C05456=1021.407,257.153,370.993,169.626,49.435,159.469
C05457=1021.401,256.905,371.022,169.622,49.439,159.470
C05458=1021.394,256.657,371.050,169.618,49.443,159.470
C05459=1021.388,256.409,371.079,169.613,49.447,159.470
C05460=1021.381,256.160,371.108,169.610,49.452,159.470
C05461=1021.375,255.912,371.135,169.605,49.456,159.471
C05462=1021.369,255.664,371.165,169.601,49.460,159.471
C05463=1021.362,255.416,371.194,169.596,49.464,159.471
C05464=1021.356,255.167,371.221,169.592,49.469,159.471
C05465=1021.349,254.919,371.250,169.588,49.473,159.472
C05466=1021.343,254.670,371.279,169.583,49.477,159.472
C05467=1021.337,254.422,371.308,169.580,49.481,159.472
C05468=1021.330,254.174,371.335,169.575,49.486,159.473
C05469=1021.324,253.926,371.364,169.571,49.490,159.473
C05470=1021.318,253.677,371.393,169.567,49.494,159.473
C05471=1021.311,253.429,371.421,169.563,49.499,159.474
C05472=1021.305,253.180,371.450,169.559,49.503,159.474
C05473=1021.299,252.932,371.479,169.555,49.507,159.474
C05474=1021.292,252.684,371.506,169.550,49.511,159.474
C05475=1021.286,252.436,371.535,169.546,49.516,159.475
C05476=1021.280,252.187,371.564,169.542,49.520,159.475
C05477=1021.273,251.939,371.592,169.538,49.524,159.475
C05478=1021.267,251.690,371.620,169.534,49.529,159.476
C05479=1021.262,251.442,371.648,169.530,49.533,159.476
C05480=1021.255,251.195,371.677,169.525,49.538,159.476
C05481=1021.249,250.946,371.705,169.522,49.542,159.477
C05482=1021.243,250.698,371.734,169.517,49.547,159.477
C05483=1021.236,250.449,371.762,169.513,49.551,159.477
C05484=1021.230,250.200,371.790,169.509,49.555,159.477
C05485=1021.224,249.952,371.819,169.504,49.560,159.478
C05486=1021.218,249.705,371.847,169.501,49.564,159.478
C05487=1021.212,249.489,371.872,169.497,49.568,159.478
C05488=1021.208,249.274,371.896,169.493,49.572,159.479
C05489=1021.202,249.058,371.920,169.490,49.575,159.479
C05490=1021.197,248.843,371.945,169.487,49.579,159.479
C05491=1021.191,248.629,371.970,169.483,49.583,159.479
C05492=1021.186,248.413,371.994,169.479,49.587,159.480
C05493=1021.180,248.198,372.018,169.475,49.591,159.480
C05494=1021.175,247.983,372.043,169.473,49.595,159.480
C05495=1021.169,247.734,372.071,169.468,49.599,159.481
C05496=1021.163,247.485,372.099,169.464,49.604,159.481
C05497=1021.156,247.237,372.128,169.460,49.608,159.481
C05498=1021.151,246.989,372.156,169.456,49.612,159.482
C05499=1021.144,246.741,372.184,169.452,49.617,159.482
C05500=1021.138,246.492,372.212,169.448,49.621,159.482
C05501=1021.133,246.243,372.240,169.443,49.626,159.483
C05502=1021.126,245.996,372.268,169.440,49.630,159.483
C05503=1021.120,245.747,372.297,169.435,49.635,159.483
C05504=1021.114,245.499,372.325,169.432,49.640,159.484
C05505=1021.108,245.251,372.352,169.427,49.644,159.484
C05506=1021.102,245.002,372.381,169.424,49.648,159.484
C05507=1021.096,244.753,372.409,169.419,49.653,159.485
C05508=1021.090,244.506,372.436,169.415,49.657,159.485
C05509=1021.084,244.257,372.465,169.411,49.662,159.485
C05510=1021.078,244.008,372.493,169.408,49.667,159.486
C05511=1021.072,243.761,372.521,169.403,49.671,159.486
C05512=1021.066,243.512,372.549,169.399,49.676,159.486
C05513=1021.060,243.263,372.577,169.395,49.681,159.487
C05514=1021.054,243.015,372.605,169.392,49.685,159.487
C05515=1021.048,242.767,372.632,169.387,49.690,159.487
C05516=1021.041,242.518,372.660,169.383,49.695,159.488
C05517=1021.036,242.270,372.688,169.379,49.699,159.488
C05518=1021.029,242.022,372.716,169.375,49.704,159.489
C05519=1021.023,241.773,372.744,169.371,49.709,159.489
C05520=1021.017,241.525,372.771,169.367,49.713,159.489
C05521=1021.010,241.277,372.799,169.364,49.718,159.490
C05522=1021.005,241.028,372.827,169.359,49.723,159.490
C05523=1020.998,240.780,372.854,169.355,49.728,159.491
C05524=1020.992,240.531,372.882,169.351,49.732,159.491
C05525=1020.986,240.283,372.910,169.347,49.737,159.491
C05526=1020.980,240.035,372.937,169.343,49.742,159.492
C05527=1020.973,239.786,372.964,169.339,49.746,159.492
C05528=1020.968,239.538,372.992,169.336,49.751,159.493
C05529=1020.961,239.289,373.020,169.331,49.756,159.493
C05530=1020.955,239.042,373.048,169.327,49.761,159.493
C05531=1020.949,238.793,373.075,169.324,49.766,159.494
C05532=1020.942,238.544,373.102,169.319,49.771,159.494
C05533=1020.937,238.295,373.130,169.316,49.776,159.495
C05534=1020.931,238.047,373.157,169.311,49.780,159.495
C05535=1020.924,237.799,373.185,169.307,49.785,159.496
C05536=1020.918,237.550,373.212,169.304,49.790,159.496
C05537=1020.911,237.302,373.239,169.299,49.795,159.496
C05538=1020.906,237.053,373.266,169.296,49.800,159.497
C05539=1020.899,236.805,373.294,169.292,49.805,159.497
C05540=1020.893,236.557,373.320,169.287,49.810,159.498
C05541=1020.886,236.308,373.348,169.284,49.815,159.498
C05542=1020.881,236.059,373.375,169.280,49.820,159.499
C05543=1020.875,235.811,373.403,169.275,49.825,159.499
C05544=1020.869,235.563,373.430,169.272,49.830,159.499
C05545=1020.862,235.314,373.457,169.268,49.835,159.500
C05546=1020.857,235.066,373.484,169.264,49.840,159.500
C05547=1020.851,234.847,373.508,169.261,49.844,159.501
C05548=1020.845,234.629,373.532,169.257,49.848,159.501
C05549=1020.840,234.410,373.556,169.254,49.853,159.502
C05550=1020.834,234.192,373.579,169.251,49.858,159.502
C05551=1020.828,233.974,373.604,169.247,49.862,159.502
C05552=1020.823,233.756,373.627,169.243,49.866,159.503
C05553=1020.818,233.537,373.652,169.240,49.871,159.503
C05554=1020.813,233.319,373.675,169.237,49.875,159.504
C05555=1020.807,233.070,373.702,169.232,49.881,159.504
C05556=1020.800,232.822,373.730,169.229,49.885,159.504
C05557=1020.794,232.574,373.756,169.225,49.890,159.505
C05558=1020.788,232.324,373.783,169.220,49.895,159.505
C05559=1020.782,232.077,373.811,169.217,49.900,159.506
C05560=1020.776,231.828,373.838,169.213,49.906,159.506
C05561=1020.770,231.579,373.864,169.209,49.911,159.507
C05562=1020.763,231.330,373.891,169.206,49.916,159.507
C05563=1020.757,231.083,373.919,169.201,49.921,159.508
C05564=1020.752,230.834,373.945,169.198,49.926,159.508
C05565=1020.745,230.585,373.973,169.194,49.931,159.509
C05566=1020.739,230.337,374.000,169.189,49.936,159.509
C05567=1020.733,230.088,374.027,169.186,49.941,159.510
C05568=1020.727,229.840,374.054,169.182,49.946,159.510
C05569=1020.721,229.592,374.080,169.178,49.952,159.511
C05570=1020.715,229.342,374.107,169.175,49.957,159.511
C05571=1020.708,229.095,374.134,169.171,49.962,159.512
C05572=1020.702,228.847,374.161,169.167,49.968,159.512
C05573=1020.696,228.598,374.188,169.163,49.973,159.513
C05574=1020.690,228.349,374.214,169.159,49.978,159.513
C05575=1020.684,228.101,374.241,169.155,49.983,159.514
C05576=1020.678,227.852,374.268,169.152,49.988,159.514
C05577=1020.672,227.604,374.295,169.148,49.994,159.515
C05578=1020.666,227.354,374.322,169.143,49.999,159.515
C05579=1020.659,227.106,374.348,169.140,50.004,159.516
C05580=1020.653,226.858,374.374,169.136,50.009,159.516
C05581=1020.648,226.610,374.401,169.132,50.015,159.517
C05582=1020.641,226.361,374.428,169.129,50.020,159.517
C05583=1020.635,226.113,374.454,169.125,50.025,159.518
C05584=1020.629,225.864,374.481,169.120,50.031,159.518
C05585=1020.622,225.615,374.507,169.117,50.037,159.519
C05586=1020.616,225.367,374.534,169.113,50.042,159.520
C05587=1020.610,225.119,374.560,169.109,50.047,159.520
C05588=1020.603,224.870,374.587,169.105,50.053,159.521
C05589=1020.598,224.622,374.613,169.101,50.058,159.521
C05590=1020.592,224.373,374.639,169.098,50.063,159.522
C05591=1020.585,224.124,374.666,169.094,50.068,159.522
C05592=1020.579,223.876,374.692,169.090,50.074,159.523
C05593=1020.573,223.627,374.719,169.086,50.080,159.523
C05594=1020.567,223.379,374.745,169.083,50.085,159.524
C05595=1020.560,223.130,374.772,169.079,50.091,159.524
C05596=1020.554,222.881,374.798,169.075,50.096,159.525
C05597=1020.549,222.633,374.824,169.071,50.102,159.526
C05598=1020.541,222.384,374.851,169.068,50.107,159.526
C05599=1020.536,222.136,374.877,169.063,50.112,159.527
C05600=1020.530,221.888,374.904,169.060,50.118,159.527
C05601=1020.524,221.639,374.929,169.057,50.123,159.528
C05602=1020.518,221.391,374.956,169.053,50.129,159.528
C05603=1020.512,221.141,374.983,169.049,50.135,159.529
C05604=1020.505,220.893,375.009,169.045,50.141,159.530
C05605=1020.500,220.644,375.035,169.042,50.146,159.530
C05606=1020.493,220.396,375.061,169.037,50.151,159.531
C05607=1020.488,220.174,375.085,169.034,50.156,159.531
C05608=1020.482,219.951,375.109,169.031,50.161,159.532
C05609=1020.477,219.729,375.132,169.027,50.166,159.532
C05610=1020.471,219.507,375.155,169.024,50.171,159.533
C05611=1020.466,219.284,375.178,169.020,50.176,159.533
C05612=1020.461,219.061,375.202,169.017,50.181,159.534
C05613=1020.455,218.838,375.226,169.014,50.186,159.534
C05614=1020.450,218.616,375.249,169.011,50.191,159.535
C05615=1020.443,218.368,375.275,169.007,50.196,159.535
C05616=1020.438,218.119,375.301,169.003,50.202,159.536
C05617=1020.431,217.871,375.327,168.999,50.208,159.537
C05618=1020.425,217.623,375.353,168.996,50.213,159.537
C05619=1020.419,217.374,375.379,168.992,50.219,159.538
C05620=1020.412,217.125,375.405,168.988,50.225,159.538
C05621=1020.406,216.877,375.431,168.984,50.231,159.539
C05622=1020.400,216.628,375.457,168.980,50.237,159.540
C05623=1020.394,216.380,375.483,168.977,50.243,159.540
C05624=1020.388,216.131,375.508,168.974,50.248,159.541
C05625=1020.382,215.882,375.534,168.970,50.254,159.541
C05626=1020.376,215.634,375.560,168.966,50.260,159.542
C05627=1020.369,215.385,375.586,168.962,50.266,159.543
C05628=1020.363,215.136,375.613,168.958,50.272,159.543
C05629=1020.357,214.888,375.638,168.954,50.277,159.544
C05630=1020.351,214.639,375.663,168.951,50.283,159.545
C05631=1020.344,214.391,375.689,168.947,50.289,159.545
C05632=1020.339,214.142,375.715,168.944,50.295,159.546
C05633=1020.333,213.893,375.741,168.940,50.301,159.547
C05634=1020.326,213.645,375.767,168.936,50.306,159.547
C05635=1020.321,213.396,375.793,168.932,50.312,159.548
C05636=1020.314,213.148,375.818,168.929,50.318,159.548
C05637=1020.308,212.900,375.844,168.925,50.324,159.549
C05638=1020.302,212.651,375.870,168.922,50.330,159.550
C05639=1020.296,212.402,375.895,168.918,50.336,159.550
C05640=1020.290,212.154,375.921,168.914,50.341,159.551
C05641=1020.284,211.905,375.947,168.910,50.347,159.551
C05642=1020.278,211.656,375.973,168.907,50.353,159.552
C05643=1020.272,211.408,375.998,168.903,50.359,159.553
C05644=1020.265,211.159,376.024,168.900,50.365,159.553
C05645=1020.260,210.910,376.050,168.896,50.371,159.554
C05646=1020.254,210.662,376.075,168.892,50.377,159.555
C05647=1020.247,210.413,376.101,168.888,50.383,159.555
C05648=1020.242,210.165,376.127,168.885,50.389,159.556
C05649=1020.235,209.916,376.153,168.882,50.395,159.557
C05650=1020.229,209.667,376.178,168.878,50.401,159.557
C05651=1020.223,209.419,376.203,168.874,50.407,159.558
C05652=1020.217,209.170,376.229,168.870,50.413,159.559
C05653=1020.211,208.921,376.254,168.867,50.419,159.559
C05654=1020.204,208.673,376.279,168.863,50.425,159.560
C05655=1020.199,208.424,376.305,168.859,50.431,159.561
C05656=1020.193,208.175,376.331,168.855,50.437,159.561
C05657=1020.186,207.927,376.357,168.852,50.443,159.562
C05658=1020.180,207.678,376.382,168.849,50.449,159.563
C05659=1020.174,207.430,376.407,168.845,50.455,159.564
C05660=1020.168,207.181,376.433,168.841,50.461,159.564
C05661=1020.161,206.932,376.458,168.838,50.468,159.565
C05662=1020.155,206.684,376.483,168.834,50.474,159.566
C05663=1020.149,206.398,376.512,168.830,50.481,159.566
C05664=1020.141,206.111,376.541,168.825,50.488,159.567
C05665=1020.134,205.825,376.571,168.821,50.495,159.568
C05666=1020.127,205.539,376.599,168.818,50.502,159.569
C05667=1020.118,205.137,376.640,168.811,50.512,159.570
C05668=1020.107,204.735,376.680,168.805,50.522,159.571
C05669=1020.097,204.333,376.721,168.800,50.532,159.572
C05670=1020.088,203.931,376.762,168.794,50.542,159.573
C05671=1020.065,202.891,376.861,168.342,50.448,159.476
C05672=1020.060,202.642,376.884,168.337,50.455,159.477
C05673=1020.055,202.393,376.907,168.333,50.463,159.478
C05674=1020.050,202.145,376.932,168.329,50.470,159.479
C05675=1020.044,201.896,376.955,168.324,50.477,159.479
C05676=1020.039,201.647,376.978,168.320,50.484,159.480
C05677=1020.034,201.398,377.002,168.316,50.492,159.481
C05678=1020.028,201.149,377.025,168.311,50.499,159.482
C05679=1020.023,200.900,377.049,168.307,50.506,159.482
C05680=1020.019,200.652,377.072,168.302,50.513,159.483
C05681=1020.013,200.403,377.096,168.298,50.520,159.484
C05682=1020.008,200.154,377.119,168.294,50.528,159.485
C05683=1020.003,199.905,377.143,168.289,50.535,159.485
C05684=1019.998,199.656,377.166,168.285,50.542,159.486
C05685=1019.992,199.407,377.189,168.280,50.549,159.487
C05686=1019.988,199.158,377.212,168.276,50.557,159.488
C05687=1019.982,198.909,377.235,168.272,50.564,159.488
C05688=1019.976,198.660,377.258,168.267,50.571,159.489
C05689=1019.971,198.411,377.282,168.263,50.579,159.490
C05690=1019.965,198.162,377.305,168.259,50.586,159.491
C05691=1019.960,197.913,377.328,168.255,50.593,159.491
C05692=1019.955,197.665,377.351,168.251,50.601,159.492
C05693=1019.950,197.416,377.374,168.246,50.608,159.493
C05694=1019.944,197.167,377.397,168.242,50.615,159.494
C05695=1019.939,196.918,377.420,168.238,50.623,159.495
C05696=1019.934,196.670,377.443,168.233,50.630,159.495
C05697=1019.928,196.421,377.466,168.229,50.637,159.496
C05698=1019.923,196.172,377.489,168.225,50.645,159.497
C05699=1019.917,195.923,377.512,168.220,50.652,159.498
C05700=1019.912,195.675,377.535,168.216,50.659,159.498
C05701=1019.907,195.425,377.558,168.212,50.667,159.499
C05702=1019.901,195.176,377.581,168.207,50.674,159.500
C05703=1019.896,194.927,377.604,168.203,50.681,159.501
C05704=1019.892,194.678,377.627,168.199,50.689,159.502
C05705=1019.886,194.429,377.650,168.195,50.696,159.502
C05706=1019.880,194.181,377.673,168.190,50.704,159.503
C05707=1019.876,193.932,377.696,168.186,50.711,159.504
C05708=1019.870,193.683,377.719,168.182,50.718,159.505
C05709=1019.865,193.434,377.741,168.178,50.726,159.505
C05710=1019.860,193.184,377.765,168.173,50.733,159.506
C05711=1019.854,192.936,377.787,168.169,50.740,159.507
C05712=1019.849,192.687,377.810,168.165,50.748,159.508
C05713=1019.844,192.439,377.833,168.160,50.755,159.508
C05714=1019.839,192.189,377.855,168.156,50.763,159.509
C05715=1019.833,191.940,377.878,168.152,50.770,159.510
C05716=1019.829,191.692,377.902,168.148,50.777,159.511
C05717=1019.823,191.442,377.924,168.144,50.785,159.512
C05718=1019.818,191.194,377.947,168.139,50.792,159.512
C05719=1019.813,190.945,377.970,168.135,50.800,159.513
C05720=1019.808,190.696,377.993,168.132,50.806,159.514
C05721=1019.803,190.447,378.015,168.127,50.814,159.515
C05722=1019.798,190.198,378.038,168.123,50.821,159.516
C05723=1019.792,189.949,378.061,168.119,50.828,159.516
C05724=1019.787,189.700,378.083,168.115,50.836,159.517
C05725=1019.782,189.451,378.107,168.110,50.843,159.518
C05726=1019.777,189.203,378.129,168.106,50.851,159.519
C05727=1019.772,188.953,378.151,168.102,50.858,159.520
C05728=1019.767,188.705,378.175,168.098,50.866,159.520
C05729=1019.762,188.455,378.197,168.094,50.872,159.521
C05730=1019.757,188.207,378.219,168.090,50.880,159.522
C05731=1019.751,187.958,378.242,168.086,50.887,159.523
C05732=1019.746,187.677,378.268,168.081,50.896,159.524
C05733=1019.740,187.396,378.294,168.077,50.904,159.525
C05734=1019.734,187.114,378.319,168.072,50.912,159.525
C05735=1019.728,186.833,378.344,168.068,50.921,159.526
C05736=1019.724,186.585,378.368,168.063,50.928,159.527
C05737=1019.718,186.335,378.390,168.059,50.935,159.528
C05738=1019.713,186.087,378.412,168.056,50.943,159.529
C05739=1019.708,185.837,378.435,168.052,50.950,159.529
C05740=1019.703,185.589,378.458,168.047,50.957,159.530
C05741=1019.698,185.339,378.480,168.043,50.965,159.531
C05742=1019.693,185.091,378.503,168.039,50.972,159.532
C05743=1019.689,184.842,378.525,168.036,50.980,159.533
C05744=1019.683,184.593,378.548,168.031,50.987,159.533
C05745=1019.678,184.344,378.570,168.027,50.994,159.534
C05746=1019.673,184.095,378.593,168.023,51.002,159.535
C05747=1019.668,183.846,378.615,168.020,51.009,159.536
C05748=1019.663,183.597,378.638,168.016,51.017,159.537
C05749=1019.658,183.348,378.661,168.011,51.024,159.537
C05750=1019.654,183.100,378.683,168.007,51.031,159.538
C05751=1019.648,182.850,378.705,168.004,51.039,159.539
C05752=1019.644,182.602,378.728,168.000,51.046,159.540
C05753=1019.638,182.352,378.750,167.996,51.054,159.541
C05754=1019.634,182.103,378.772,167.991,51.061,159.541
C05755=1019.628,181.854,378.794,167.988,51.068,159.542
C05756=1019.623,181.605,378.817,167.984,51.076,159.543
C05757=1019.617,181.356,378.839,167.980,51.083,159.544
C05758=1019.612,181.107,378.860,167.976,51.091,159.545
C05759=1019.607,180.858,378.883,167.972,51.098,159.546
C05760=1019.601,180.609,378.904,167.968,51.106,159.547
C05761=1019.596,180.361,378.926,167.964,51.114,159.547
C05762=1019.591,180.111,378.948,167.960,51.122,159.548
C05763=1019.585,179.863,378.969,167.957,51.129,159.549
C05764=1019.580,179.613,378.991,167.953,51.137,159.550
C05765=1019.575,179.364,379.013,167.949,51.145,159.551
C05766=1019.569,179.116,379.035,167.944,51.152,159.552
C05767=1019.564,178.866,379.057,167.940,51.160,159.553
C05768=1019.559,178.617,379.079,167.936,51.168,159.553
C05769=1019.554,178.369,379.100,167.932,51.176,159.554
C05770=1019.548,178.119,379.122,167.929,51.182,159.555
C05771=1019.544,177.870,379.143,167.925,51.190,159.556
C05772=1019.538,177.621,379.165,167.921,51.198,159.557
C05773=1019.533,177.372,379.187,167.917,51.205,159.558
C05774=1019.528,177.123,379.209,167.913,51.213,159.559
C05775=1019.522,176.875,379.230,167.909,51.221,159.559
C05776=1019.517,176.625,379.252,167.906,51.229,159.561
C05777=1019.512,176.376,379.274,167.902,51.236,159.561
C05778=1019.506,176.128,379.295,167.898,51.244,159.562
C05779=1019.501,175.878,379.318,167.894,51.252,159.563
C05780=1019.496,175.629,379.338,167.889,51.259,159.564
C05781=1019.491,175.380,379.360,167.887,51.267,159.565
C05782=1019.486,175.131,379.382,167.883,51.275,159.566
C05783=1019.480,174.882,379.403,167.879,51.282,159.566
C05784=1019.475,174.634,379.425,167.874,51.290,159.567
C05785=1019.470,174.385,379.447,167.871,51.297,159.568
C05786=1019.464,174.135,379.468,167.868,51.305,159.569
C05787=1019.460,173.886,379.490,167.863,51.312,159.570
C05788=1019.455,173.637,379.512,167.859,51.320,159.571
C05789=1019.449,173.389,379.533,167.856,51.328,159.572
C05790=1019.444,173.139,379.555,167.852,51.336,159.573
C05791=1019.439,172.890,379.577,167.848,51.343,159.573
C05792=1019.434,172.641,379.598,167.844,51.351,159.574
C05793=1019.429,172.392,379.620,167.841,51.359,159.575
C05794=1019.423,172.143,379.641,167.837,51.366,159.576
C05795=1019.418,171.894,379.662,167.833,51.374,159.577
C05796=1019.412,171.612,379.687,167.830,51.382,159.578
C05797=1019.407,171.331,379.711,167.825,51.391,159.579
C05798=1019.401,171.050,379.735,167.820,51.400,159.580
C05799=1019.395,170.768,379.759,167.817,51.408,159.581
C05800=1019.390,170.519,379.781,167.813,51.416,159.582
C05801=1019.386,170.270,379.802,167.808,51.423,159.582
C05802=1019.380,170.021,379.824,167.805,51.431,159.583
C05803=1019.375,169.771,379.846,167.802,51.439,159.584
C05804=1019.370,169.522,379.867,167.797,51.446,159.585
C05805=1019.365,169.274,379.888,167.794,51.454,159.586
C05806=1019.360,169.025,379.910,167.790,51.462,159.587
C05807=1019.354,168.776,379.931,167.787,51.470,159.588
C05808=1019.350,168.527,379.953,167.783,51.477,159.589
C05809=1019.345,168.277,379.974,167.779,51.484,159.589
C05810=1019.340,168.029,379.995,167.775,51.492,159.590
C05811=1019.334,167.779,380.017,167.772,51.499,159.591
C05812=1019.330,167.530,380.038,167.768,51.507,159.592
C05813=1019.324,167.281,380.060,167.764,51.515,159.593
C05814=1019.320,167.032,380.081,167.761,51.522,159.594
C05815=1019.314,166.783,380.102,167.757,51.530,159.595
C05816=1019.309,166.534,380.123,167.754,51.538,159.596
C05817=1019.305,166.285,380.145,167.750,51.545,159.596
C05818=1019.299,166.036,380.166,167.746,51.553,159.597
C05819=1019.295,165.787,380.188,167.743,51.561,159.598
C05820=1019.290,165.538,380.209,167.739,51.568,159.599
C05821=1019.284,165.289,380.230,167.736,51.575,159.600
C05822=1019.280,165.040,380.251,167.732,51.583,159.601
C05823=1019.274,164.791,380.272,167.728,51.591,159.602
C05824=1019.270,164.542,380.294,167.725,51.598,159.603
C05825=1019.265,164.293,380.315,167.721,51.606,159.603
C05826=1019.260,164.044,380.336,167.718,51.614,159.604
C05827=1019.255,163.795,380.358,167.714,51.621,159.605
C05828=1019.249,163.545,380.379,167.711,51.629,159.606
C05829=1019.244,163.297,380.401,167.707,51.637,159.607
C05830=1019.240,163.047,380.422,167.703,51.644,159.608
C05831=1019.234,162.799,380.443,167.700,51.652,159.609
C05832=1019.230,162.550,380.464,167.696,51.660,159.610
C05833=1019.226,162.300,380.485,167.693,51.667,159.610
C05834=1019.220,162.052,380.506,167.689,51.675,159.611
C05835=1019.216,161.803,380.527,167.686,51.682,159.612
C05836=1019.210,161.554,380.549,167.682,51.690,159.613
C05837=1019.206,161.305,380.570,167.679,51.697,159.614
C05838=1019.201,161.055,380.591,167.675,51.704,159.615
C05839=1019.196,160.807,380.612,167.672,51.712,159.616
C05840=1019.191,160.557,380.633,167.668,51.720,159.617
C05841=1019.186,160.308,380.654,167.665,51.727,159.617
C05842=1019.181,160.059,380.676,167.661,51.735,159.618
C05843=1019.176,159.810,380.697,167.658,51.743,159.619
C05844=1019.171,159.561,380.717,167.654,51.750,159.620
C05845=1019.166,159.312,380.739,167.651,51.758,159.621
C05846=1019.161,159.063,380.760,167.647,51.766,159.622
C05847=1019.157,158.813,380.781,167.644,51.773,159.623
C05848=1019.151,158.564,380.802,167.640,51.781,159.624
C05849=1019.146,158.315,380.822,167.637,51.789,159.625
C05850=1019.142,158.066,380.843,167.634,51.796,159.626
C05851=1019.137,157.817,380.863,167.630,51.804,159.626
C05852=1019.131,157.569,380.885,167.627,51.812,159.627
C05853=1019.126,157.320,380.905,167.623,51.820,159.628
C05854=1019.121,157.070,380.926,167.619,51.827,159.629
C05855=1019.116,156.821,380.946,167.616,51.835,159.630
C05856=1019.110,156.572,380.967,167.612,51.843,159.631
C05857=1019.106,156.323,380.988,167.610,51.851,159.632
C05858=1019.101,156.074,381.009,167.606,51.859,159.633
C05859=1019.095,155.825,381.029,167.602,51.867,159.634
C05860=1019.090,155.543,381.052,167.598,51.875,159.635
C05861=1019.084,155.261,381.076,167.595,51.884,159.636
C05862=1019.078,154.978,381.099,167.590,51.892,159.637
C05863=1019.072,154.697,381.122,167.587,51.901,159.638
C05864=1019.067,154.448,381.142,167.583,51.909,159.639
C05865=1019.062,154.199,381.163,167.580,51.917,159.640
C05866=1019.057,153.950,381.184,167.576,51.925,159.641
C05867=1019.052,153.701,381.205,167.574,51.933,159.642
C05868=1019.047,153.452,381.225,167.570,51.941,159.643
C05869=1019.042,153.202,381.245,167.566,51.949,159.644
C05870=1019.037,152.953,381.265,167.563,51.956,159.644
C05871=1019.032,152.704,381.286,167.559,51.964,159.645
C05872=1019.027,152.455,381.306,167.556,51.971,159.646
C05873=1019.021,152.206,381.327,167.552,51.979,159.647
C05874=1019.016,151.957,381.347,167.549,51.987,159.648
C05875=1019.012,151.708,381.367,167.546,51.995,159.649
C05876=1019.007,151.459,381.387,167.543,52.003,159.650
C05877=1019.001,151.209,381.408,167.539,52.011,159.651
C05878=1018.996,150.960,381.429,167.535,52.019,159.652
C05879=1018.991,150.711,381.449,167.532,52.027,159.653
C05880=1018.986,150.462,381.469,167.529,52.035,159.654
C05881=1018.981,150.213,381.489,167.525,52.042,159.655
C05882=1018.976,149.964,381.510,167.522,52.050,159.655
C05883=1018.971,149.715,381.530,167.519,52.057,159.656
C05884=1018.966,149.465,381.550,167.515,52.065,159.657
C05885=1018.961,149.217,381.570,167.512,52.073,159.658
C05886=1018.956,148.968,381.591,167.509,52.081,159.659
C05887=1018.951,148.718,381.611,167.506,52.089,159.660
C05888=1018.946,148.469,381.631,167.502,52.097,159.661
C05889=1018.941,148.220,381.651,167.499,52.105,159.662
C05890=1018.936,147.971,381.672,167.495,52.113,159.663
C05891=1018.931,147.721,381.692,167.493,52.120,159.664
C05892=1018.925,147.473,381.712,167.488,52.128,159.665
C05893=1018.920,147.223,381.731,167.486,52.135,159.666
C05894=1018.915,146.974,381.752,167.482,52.144,159.667
C05895=1018.910,146.725,381.772,167.479,52.151,159.668
C05896=1018.905,146.475,381.792,167.475,52.159,159.669
C05897=1018.900,146.227,381.812,167.473,52.167,159.670
C05898=1018.895,145.977,381.832,167.469,52.175,159.671
C05899=1018.890,145.728,381.853,167.466,52.183,159.672
C05900=1018.885,145.480,381.873,167.462,52.191,159.672
C05901=1018.880,145.230,381.892,167.460,52.199,159.673
C05902=1018.874,144.981,381.913,167.456,52.207,159.674
C05903=1018.870,144.731,381.933,167.453,52.214,159.675
C05904=1018.864,144.483,381.952,167.449,52.222,159.676
C05905=1018.859,144.234,381.972,167.446,52.231,159.677
C05906=1018.854,143.984,381.992,167.443,52.238,159.678
C05907=1018.849,143.736,382.011,167.439,52.246,159.679
C05908=1018.844,143.486,382.031,167.436,52.254,159.680
C05909=1018.839,143.237,382.052,167.433,52.262,159.681
C05910=1018.834,142.988,382.071,167.430,52.270,159.682
C05911=1018.828,142.739,382.091,167.426,52.278,159.683
C05912=1018.823,142.489,382.111,167.423,52.286,159.684
C05913=1018.819,142.240,382.131,167.420,52.294,159.685
C05914=1018.813,141.991,382.150,167.417,52.302,159.686
C05915=1018.808,141.742,382.170,167.413,52.310,159.687
C05916=1018.803,141.493,382.191,167.410,52.317,159.688
C05917=1018.798,141.244,382.210,167.407,52.325,159.689
C05918=1018.793,140.994,382.230,167.404,52.333,159.690
C05919=1018.788,140.746,382.250,167.401,52.341,159.691
C05920=1018.782,140.496,382.269,167.397,52.349,159.692
C05921=1018.777,140.247,382.289,167.395,52.357,159.693
C05922=1018.773,139.998,382.309,167.391,52.365,159.694
C05923=1018.768,139.748,382.329,167.388,52.373,159.695
C05924=1018.761,139.386,382.357,167.383,52.384,159.696
C05925=1018.753,139.023,382.386,167.379,52.396,159.697
C05926=1018.745,138.661,382.415,167.373,52.407,159.698
C05927=1018.738,138.298,382.443,167.369,52.418,159.700
C05928=1018.733,138.048,382.463,167.366,52.426,159.701
C05929=1018.728,137.799,382.483,167.363,52.434,159.702
C05930=1018.723,137.550,382.502,167.360,52.442,159.703
C05931=1018.718,137.301,382.522,167.356,52.450,159.704
C05932=1018.713,137.052,382.541,167.353,52.458,159.705
C05933=1018.708,136.802,382.561,167.350,52.466,159.706
C05934=1018.703,136.554,382.580,167.347,52.474,159.707
C05935=1018.698,136.304,382.600,167.343,52.482,159.708
C05936=1018.692,136.054,382.619,167.341,52.490,159.709
C05937=1018.688,135.805,382.639,167.337,52.498,159.710
C05938=1018.682,135.556,382.659,167.334,52.506,159.711
C05939=1018.677,135.307,382.678,167.332,52.513,159.712
C05940=1018.672,135.058,382.697,167.328,52.522,159.713
C05941=1018.667,134.809,382.717,167.325,52.529,159.714
C05942=1018.662,134.560,382.736,167.321,52.537,159.714
C05943=1018.657,134.311,382.755,167.319,52.546,159.716
C05944=1018.648,133.893,382.788,167.313,52.559,159.717
C05945=1018.639,133.475,382.820,167.308,52.572,159.719
C05946=1018.631,133.057,382.852,167.303,52.586,159.720
C05947=1018.623,132.640,382.885,167.297,52.599,159.722
C05948=1018.617,132.391,382.904,167.294,52.607,159.723
C05949=1018.613,132.142,382.924,167.292,52.615,159.724
C05950=1018.607,131.892,382.943,167.288,52.623,159.725
C05951=1018.602,131.643,382.962,167.286,52.631,159.726
C05952=1018.597,131.394,382.982,167.282,52.639,159.727
C05953=1018.592,131.145,383.000,167.279,52.647,159.728
C05954=1018.587,130.895,383.020,167.276,52.655,159.729
C05955=1018.582,130.646,383.039,167.273,52.663,159.730
C05956=1018.576,130.397,383.058,167.270,52.671,159.731
C05957=1018.572,130.148,383.078,167.267,52.679,159.732
C05958=1018.566,129.899,383.097,167.264,52.687,159.733
C05959=1018.562,129.650,383.117,167.260,52.695,159.734
C05960=1018.556,129.400,383.136,167.258,52.703,159.735
C05961=1018.552,129.151,383.154,167.254,52.711,159.736
C05962=1018.546,128.901,383.173,167.251,52.719,159.737
C05963=1018.541,128.653,383.192,167.248,52.727,159.738
C05964=1018.536,128.404,383.211,167.245,52.735,159.739
C05965=1018.530,128.154,383.229,167.242,52.744,159.740
C05966=1018.525,127.905,383.248,167.239,52.751,159.741
C05967=1018.520,127.656,383.268,167.235,52.760,159.742
C05968=1018.514,127.407,383.286,167.233,52.767,159.743
C05969=1018.509,127.157,383.305,167.229,52.776,159.744
C05970=1018.504,126.908,383.324,167.227,52.784,159.745
C05971=1018.499,126.658,383.344,167.223,52.792,159.746
C05972=1018.494,126.409,383.362,167.221,52.800,159.747
C05973=1018.489,126.160,383.381,167.217,52.808,159.748
C05974=1018.483,125.911,383.400,167.214,52.816,159.749
C05975=1018.479,125.661,383.418,167.212,52.824,159.750
C05976=1018.473,125.412,383.437,167.209,52.833,159.751
C05977=1018.468,125.163,383.456,167.206,52.841,159.752
C05978=1018.463,124.914,383.474,167.202,52.849,159.753
C05979=1018.457,124.665,383.494,167.200,52.857,159.754
C05980=1018.452,124.416,383.513,167.196,52.865,159.755
C05981=1018.447,124.166,383.531,167.193,52.873,159.756
C05982=1018.442,123.917,383.550,167.190,52.881,159.757
C05983=1018.437,123.668,383.569,167.187,52.889,159.758
C05984=1018.431,123.386,383.590,167.184,52.898,159.759
C05985=1018.425,123.104,383.611,167.180,52.908,159.760
C05986=1018.419,122.822,383.632,167.177,52.916,159.761
C05987=1018.414,122.540,383.654,167.174,52.925,159.762
C05988=1018.409,122.290,383.673,167.170,52.934,159.763
C05989=1018.403,122.041,383.691,167.167,52.941,159.764
C05990=1018.399,121.792,383.710,167.165,52.950,159.766
C05991=1018.393,121.542,383.729,167.162,52.958,159.766
C05992=1018.388,121.293,383.747,167.159,52.966,159.767
C05993=1018.383,121.044,383.766,167.155,52.974,159.768
C05994=1018.377,120.795,383.785,167.153,52.982,159.769
C05995=1018.373,120.546,383.803,167.150,52.990,159.770
C05996=1018.368,120.297,383.822,167.147,52.998,159.771
C05997=1018.362,120.047,383.841,167.144,53.006,159.772
C05998=1018.357,119.798,383.860,167.140,53.014,159.773
C05999=1018.353,119.548,383.878,167.138,53.022,159.774
C06000=1018.347,119.299,383.898,167.135,53.030,159.775
C06001=1018.343,119.050,383.916,167.132,53.038,159.776
C06002=1018.338,118.801,383.935,167.129,53.046,159.777
C06003=1018.333,118.552,383.953,167.126,53.054,159.778
C06004=1018.327,118.302,383.972,167.123,53.063,159.779
C06005=1018.322,118.053,383.990,167.121,53.070,159.780
C06006=1018.317,117.804,384.009,167.117,53.079,159.781
C06007=1018.312,117.555,384.027,167.114,53.087,159.782
C06008=1018.307,117.305,384.046,167.112,53.094,159.783
C06009=1018.302,117.056,384.065,167.108,53.103,159.784
C06010=1018.297,116.807,384.084,167.106,53.111,159.785
C06011=1018.292,116.558,384.102,167.103,53.118,159.786
C06012=1018.287,116.308,384.120,167.099,53.127,159.787
C06013=1018.282,116.059,384.139,167.097,53.134,159.788
C06014=1018.277,115.810,384.157,167.094,53.142,159.789
C06015=1018.272,115.561,384.176,167.091,53.151,159.790
C06016=1018.266,115.311,384.195,167.088,53.158,159.791
C06017=1018.261,115.062,384.214,167.086,53.166,159.792
C06018=1018.256,114.813,384.232,167.082,53.175,159.793
C06019=1018.252,114.563,384.250,167.079,53.182,159.794
C06020=1018.247,114.315,384.269,167.077,53.190,159.795
C06021=1018.242,114.064,384.288,167.074,53.198,159.796
C06022=1018.237,113.815,384.306,167.071,53.206,159.797
C06023=1018.232,113.566,384.325,167.068,53.214,159.798
C06024=1018.227,113.317,384.343,167.066,53.222,159.799
C06025=1018.222,113.068,384.362,167.062,53.230,159.800
C06026=1018.217,112.819,384.380,167.059,53.238,159.801
C06027=1018.212,112.569,384.399,167.056,53.245,159.802
C06028=1018.207,112.320,384.417,167.054,53.253,159.803
C06029=1018.202,112.071,384.436,167.050,53.262,159.804
C06030=1018.197,111.822,384.453,167.048,53.270,159.805
C06031=1018.192,111.572,384.471,167.045,53.278,159.806
C06032=1018.187,111.322,384.490,167.042,53.286,159.807
C06033=1018.181,111.074,384.509,167.040,53.294,159.808
C06034=1018.176,110.824,384.526,167.036,53.302,159.809
C06035=1018.171,110.575,384.545,167.033,53.310,159.810
C06036=1018.166,110.326,384.563,167.031,53.318,159.811
C06037=1018.162,110.076,384.581,167.027,53.327,159.812
C06038=1018.155,109.827,384.599,167.025,53.334,159.813
C06039=1018.151,109.577,384.617,167.022,53.343,159.814
C06040=1018.146,109.329,384.636,167.019,53.351,159.815
C06041=1018.140,109.080,384.653,167.017,53.359,159.816
C06042=1018.135,108.830,384.672,167.013,53.367,159.817
C06043=1018.131,108.581,384.690,167.010,53.375,159.818
C06044=1018.125,108.332,384.707,167.007,53.384,159.819
C06045=1018.120,108.082,384.726,167.005,53.392,159.820
C06046=1018.114,107.833,384.743,167.002,53.400,159.821
C06047=1018.109,107.583,384.762,166.999,53.408,159.822
C06048=1018.104,107.301,384.782,166.996,53.417,159.823
C06049=1018.098,107.019,384.801,166.993,53.426,159.825
C06050=1018.092,106.737,384.822,166.990,53.436,159.826
C06051=1018.086,106.455,384.842,166.986,53.445,159.827
C06052=1018.081,106.206,384.861,166.983,53.453,159.828
C06053=1018.075,105.956,384.878,166.981,53.461,159.829
C06054=1018.071,105.707,384.896,166.977,53.470,159.830
C06055=1018.065,105.458,384.914,166.975,53.477,159.831
C06056=1018.060,105.209,384.932,166.972,53.486,159.832
C06057=1018.055,104.960,384.950,166.969,53.494,159.833
C06058=1018.050,104.710,384.968,166.967,53.502,159.834
C06059=1018.045,104.461,384.986,166.963,53.511,159.835
C06060=1018.040,104.212,385.003,166.961,53.519,159.836
C06061=1018.035,103.961,385.021,166.958,53.526,159.837
C06062=1018.029,103.712,385.039,166.955,53.535,159.838
C06063=1018.024,103.463,385.057,166.952,53.543,159.839
C06064=1018.019,103.214,385.075,166.950,53.551,159.840
C06065=1018.014,102.965,385.093,166.946,53.559,159.841
C06066=1018.009,102.715,385.110,166.944,53.568,159.842
C06067=1018.004,102.466,385.128,166.942,53.575,159.843
C06068=1017.998,102.217,385.146,166.938,53.584,159.844
C06069=1017.993,101.968,385.164,166.936,53.592,159.845
C06070=1017.989,101.718,385.182,166.933,53.600,159.846
C06071=1017.983,101.469,385.199,166.930,53.608,159.847
C06072=1017.979,101.219,385.217,166.927,53.616,159.848
C06073=1017.973,100.970,385.235,166.925,53.624,159.849
C06074=1017.968,100.721,385.253,166.921,53.632,159.850
C06075=1017.963,100.472,385.271,166.919,53.640,159.851
C06076=1017.958,100.223,385.289,166.916,53.648,159.852
C06077=1017.953,99.973,385.306,166.913,53.656,159.853
C06078=1017.948,99.724,385.324,166.910,53.664,159.854
C06079=1017.943,99.475,385.341,166.908,53.672,159.855
C06080=1017.938,99.225,385.360,166.905,53.680,159.856
C06081=1017.933,98.976,385.376,166.902,53.688,159.857
C06082=1017.928,98.726,385.395,166.900,53.697,159.859
C06083=1017.922,98.477,385.412,166.896,53.705,159.860
C06084=1017.917,98.227,385.429,166.894,53.713,159.861
C06085=1017.912,97.978,385.447,166.891,53.721,159.862
C06086=1017.907,97.729,385.465,166.888,53.730,159.863
C06087=1017.902,97.479,385.482,166.886,53.738,159.864
C06088=1017.896,97.230,385.499,166.882,53.747,159.865
C06089=1017.891,96.981,385.517,166.880,53.755,159.866
C06090=1017.886,96.731,385.534,166.877,53.763,159.867
C06091=1017.881,96.482,385.552,166.874,53.771,159.868
C06092=1017.875,96.233,385.569,166.871,53.779,159.869
C06093=1017.870,95.984,385.586,166.869,53.788,159.870
C06094=1017.865,95.734,385.604,166.866,53.796,159.871
C06095=1017.860,95.485,385.621,166.864,53.804,159.872
C06096=1017.854,95.236,385.639,166.860,53.812,159.873
C06097=1017.849,94.986,385.656,166.858,53.820,159.874
C06098=1017.845,94.737,385.673,166.855,53.828,159.875
C06099=1017.840,94.488,385.690,166.852,53.837,159.876
C06100=1017.834,94.239,385.708,166.849,53.844,159.877
C06101=1017.829,93.989,385.725,166.847,53.853,159.878
C06102=1017.824,93.740,385.743,166.844,53.862,159.879
C06103=1017.819,93.491,385.760,166.841,53.869,159.880
C06104=1017.813,93.241,385.777,166.839,53.877,159.881
C06105=1017.808,92.992,385.795,166.836,53.886,159.882
C06106=1017.803,92.742,385.812,166.833,53.894,159.883
C06107=1017.798,92.493,385.830,166.831,53.902,159.884
C06108=1017.793,92.243,385.847,166.827,53.910,159.885
C06109=1017.788,91.995,385.864,166.825,53.918,159.886
C06110=1017.783,91.745,385.881,166.822,53.926,159.887
C06111=1017.778,91.496,385.899,166.819,53.934,159.888
C06112=1017.772,91.214,385.917,166.816,53.944,159.890
C06113=1017.766,90.931,385.938,166.813,53.953,159.891
C06114=1017.760,90.650,385.957,166.810,53.962,159.892
C06115=1017.755,90.368,385.976,166.807,53.971,159.893
C06116=1017.750,90.119,385.995,166.805,53.979,159.894
C06117=1017.745,89.869,386.011,166.802,53.988,159.895
C06118=1017.739,89.619,386.028,166.799,53.996,159.896
C06119=1017.734,89.370,386.046,166.797,54.004,159.897
C06120=1017.729,89.120,386.063,166.793,54.012,159.898
C06121=1017.724,88.872,386.080,166.791,54.020,159.899
C06122=1017.719,88.622,386.097,166.789,54.028,159.900
C06123=1017.714,88.373,386.114,166.785,54.037,159.901
C06124=1017.709,88.123,386.131,166.783,54.045,159.902
C06125=1017.703,87.874,386.148,166.781,54.053,159.903
C06126=1017.697,87.625,386.165,166.777,54.062,159.904
C06127=1017.692,87.375,386.182,166.775,54.070,159.905
C06128=1017.688,87.126,386.198,166.772,54.078,159.906
C06129=1017.682,86.877,386.216,166.770,54.087,159.908
C06130=1017.677,86.627,386.233,166.767,54.095,159.909
C06131=1017.672,86.378,386.249,166.764,54.103,159.910
C06132=1017.666,86.128,386.266,166.761,54.111,159.911
C06133=1017.661,85.880,386.283,166.758,54.120,159.912
C06134=1017.656,85.630,386.300,166.756,54.128,159.913
C06135=1017.651,85.380,386.317,166.753,54.136,159.914
C06136=1017.646,85.131,386.334,166.750,54.145,159.915
C06137=1017.641,84.881,386.351,166.748,54.153,159.916
C06138=1017.636,84.632,386.367,166.746,54.161,159.917
C06139=1017.630,84.383,386.384,166.742,54.169,159.918
C06140=1017.625,84.134,386.401,166.740,54.177,159.919
C06141=1017.619,83.884,386.418,166.737,54.185,159.920
C06142=1017.614,83.634,386.435,166.734,54.194,159.921
C06143=1017.609,83.385,386.451,166.732,54.202,159.922
C06144=1017.604,83.136,386.468,166.729,54.211,159.923
C06145=1017.599,82.887,386.486,166.726,54.219,159.924
C06146=1017.594,82.637,386.503,166.724,54.227,159.925
C06147=1017.589,82.388,386.519,166.721,54.235,159.926
C06148=1017.584,82.139,386.536,166.718,54.243,159.927
C06149=1017.579,81.889,386.553,166.716,54.251,159.928
C06150=1017.573,81.639,386.570,166.712,54.260,159.929
C06151=1017.568,81.391,386.586,166.710,54.268,159.930
C06152=1017.563,81.141,386.602,166.708,54.276,159.931
C06153=1017.557,80.892,386.620,166.705,54.284,159.932
C06154=1017.552,80.642,386.637,166.702,54.292,159.933
C06155=1017.547,80.393,386.653,166.700,54.300,159.934
C06156=1017.542,80.144,386.670,166.697,54.308,159.935
C06157=1017.537,79.894,386.687,166.694,54.317,159.936
C06158=1017.532,79.645,386.704,166.692,54.325,159.937
C06159=1017.527,79.395,386.720,166.689,54.333,159.938
C06160=1017.522,79.146,386.737,166.686,54.341,159.939
C06161=1017.517,78.896,386.754,166.683,54.349,159.940
C06162=1017.511,78.647,386.770,166.681,54.357,159.941
C06163=1017.506,78.398,386.787,166.679,54.365,159.943
C06164=1017.501,78.148,386.804,166.675,54.374,159.943
C06165=1017.496,77.899,386.820,166.673,54.382,159.944
C06166=1017.491,77.649,386.837,166.671,54.390,159.946
C06167=1017.486,77.400,386.854,166.667,54.398,159.946
C06168=1017.481,77.151,386.870,166.665,54.406,159.948
C06169=1017.476,76.901,386.887,166.663,54.414,159.949
C06170=1017.470,76.652,386.903,166.660,54.423,159.950
C06171=1017.466,76.403,386.920,166.658,54.431,159.951
C06172=1017.460,76.153,386.937,166.655,54.440,159.952
C06173=1017.455,75.903,386.954,166.652,54.448,159.953
C06174=1017.450,75.655,386.970,166.650,54.456,159.954
C06175=1017.445,75.405,386.986,166.647,54.464,159.955
C06176=1017.439,75.123,387.005,166.643,54.474,159.956
C06177=1017.433,74.841,387.023,166.640,54.483,159.957
C06178=1017.427,74.559,387.042,166.638,54.492,159.958
C06179=1017.421,74.277,387.060,166.635,54.502,159.960
C06180=1017.416,74.028,387.076,166.633,54.510,159.961
C06181=1017.411,73.779,387.093,166.630,54.518,159.962
C06182=1017.405,73.529,387.109,166.627,54.526,159.963
C06183=1017.400,73.280,387.126,166.624,54.535,159.964
C06184=1017.395,73.030,387.141,166.622,54.543,159.965
C06185=1017.390,72.781,387.158,166.619,54.551,159.966
C06186=1017.385,72.532,387.175,166.616,54.559,159.967
C06187=1017.379,72.282,387.191,166.614,54.568,159.968
C06188=1017.374,72.033,387.207,166.611,54.576,159.969
C06189=1017.369,71.783,387.223,166.608,54.584,159.970
C06190=1017.364,71.535,387.239,166.606,54.592,159.971
C06191=1017.359,71.285,387.256,166.603,54.600,159.972
C06192=1017.353,71.035,387.272,166.600,54.609,159.973
C06193=1017.348,70.786,387.288,166.598,54.617,159.974
C06194=1017.343,70.536,387.305,166.596,54.625,159.975
C06195=1017.338,70.288,387.321,166.592,54.633,159.976
C06196=1017.333,70.037,387.337,166.590,54.641,159.977
C06197=1017.327,69.788,387.353,166.588,54.649,159.978
C06198=1017.322,69.539,387.370,166.585,54.658,159.979
C06199=1017.317,69.289,387.385,166.582,54.666,159.980
C06200=1017.312,69.040,387.402,166.580,54.674,159.981
C06201=1017.307,68.790,387.419,166.577,54.682,159.982
C06202=1017.302,68.541,387.434,166.574,54.691,159.983
C06203=1017.297,68.292,387.451,166.572,54.699,159.984
C06204=1017.291,68.043,387.467,166.570,54.707,159.985
C06205=1017.286,67.793,387.483,166.567,54.716,159.986
C06206=1017.280,67.543,387.499,166.565,54.724,159.988
C06207=1017.276,67.294,387.515,166.562,54.732,159.989
C06208=1017.270,67.044,387.531,166.559,54.741,159.989
C06209=1017.265,66.795,387.546,166.557,54.749,159.991
C06210=1017.260,66.545,387.563,166.553,54.757,159.991
C06211=1017.255,66.296,387.578,166.551,54.765,159.993
C06212=1017.250,66.046,387.595,166.549,54.774,159.994
C06213=1017.244,65.798,387.611,166.546,54.782,159.995
C06214=1017.239,65.548,387.627,166.543,54.790,159.996
C06215=1017.234,65.299,387.643,166.541,54.798,159.997
C06216=1017.228,65.049,387.659,166.538,54.807,159.998
C06217=1017.224,64.800,387.675,166.536,54.815,159.999
C06218=1017.218,64.550,387.691,166.533,54.823,160.000
C06219=1017.213,64.301,387.706,166.530,54.831,160.001
C06220=1017.208,64.051,387.723,166.528,54.840,160.002
C06221=1017.203,63.802,387.738,166.526,54.848,160.003
C06222=1017.198,63.552,387.755,166.522,54.856,160.004
C06223=1017.193,63.303,387.770,166.520,54.864,160.005
C06224=1017.187,63.054,387.786,166.518,54.872,160.006
C06225=1017.182,62.804,387.802,166.515,54.881,160.007
C06226=1017.177,62.554,387.817,166.512,54.889,160.008
C06227=1017.171,62.305,387.833,166.510,54.898,160.009
C06228=1017.166,62.055,387.849,166.507,54.906,160.010
C06229=1017.161,61.806,387.864,166.504,54.915,160.011
C06230=1017.155,61.556,387.880,166.502,54.923,160.012
C06231=1017.150,61.307,387.895,166.500,54.931,160.013
C06232=1017.144,61.058,387.911,166.496,54.940,160.014
C06233=1017.139,60.808,387.926,166.495,54.948,160.016
C06234=1017.133,60.558,387.942,166.491,54.957,160.016
C06235=1017.129,60.309,387.958,166.489,54.965,160.018
C06236=1017.124,60.060,387.973,166.486,54.974,160.018
C06237=1017.118,59.810,387.989,166.484,54.982,160.020
C06238=1017.113,59.561,388.004,166.480,54.990,160.020
C06239=1017.107,59.311,388.020,166.478,54.998,160.022
C06240=1017.102,59.030,388.037,166.476,55.008,160.023
C06241=1017.095,58.748,388.055,166.473,55.018,160.024
C06242=1017.089,58.465,388.073,166.469,55.027,160.025
C06243=1017.083,58.184,388.090,166.467,55.037,160.026
C06244=1017.078,57.934,388.106,166.464,55.045,160.027
C06245=1017.073,57.685,388.121,166.461,55.053,160.028
C06246=1017.067,57.435,388.136,166.459,55.061,160.029
C06247=1017.062,57.186,388.152,166.456,55.070,160.030
C06248=1017.057,56.937,388.167,166.454,55.078,160.032
C06249=1017.051,56.687,388.183,166.451,55.086,160.033
C06250=1017.046,56.438,388.198,166.448,55.095,160.034
C06251=1017.041,56.189,388.213,166.446,55.104,160.035
C06252=1017.035,55.939,388.229,166.443,55.112,160.036
C06253=1017.030,55.689,388.244,166.441,55.120,160.037
C06254=1017.025,55.440,388.260,166.439,55.128,160.038
C06255=1017.019,55.191,388.276,166.436,55.137,160.039
C06256=1017.014,54.942,388.291,166.433,55.145,160.040
C06257=1017.009,54.692,388.306,166.430,55.154,160.041
C06258=1017.004,54.442,388.321,166.428,55.162,160.042
C06259=1016.999,54.193,388.337,166.426,55.170,160.043
C06260=1016.994,53.943,388.353,166.423,55.179,160.044
C06261=1016.989,53.694,388.368,166.420,55.187,160.045
C06262=1016.984,53.444,388.383,166.418,55.195,160.046
C06263=1016.978,53.194,388.399,166.415,55.203,160.047
C06264=1016.973,52.945,388.414,166.412,55.211,160.048
C06265=1016.968,52.696,388.429,166.410,55.219,160.049
C06266=1016.962,52.446,388.445,166.407,55.228,160.050
C06267=1016.957,52.197,388.460,166.405,55.236,160.051
C06268=1016.952,51.948,388.476,166.403,55.244,160.052
C06269=1016.946,51.698,388.491,166.399,55.253,160.053
C06270=1016.941,51.449,388.506,166.397,55.261,160.054
C06271=1016.936,51.199,388.521,166.394,55.269,160.055
C06272=1016.930,50.949,388.537,166.392,55.277,160.056
C06273=1016.925,50.700,388.552,166.390,55.286,160.057
C06274=1016.920,50.451,388.567,166.388,55.294,160.058
C06275=1016.915,50.202,388.583,166.384,55.302,160.059
C06276=1016.910,49.952,388.598,166.382,55.310,160.060
C06277=1016.905,49.702,388.613,166.380,55.318,160.061
C06278=1016.900,49.453,388.628,166.376,55.327,160.062
C06279=1016.894,49.203,388.644,166.374,55.335,160.063
C06280=1016.889,48.954,388.659,166.372,55.343,160.064
C06281=1016.885,48.704,388.675,166.369,55.351,160.065
C06282=1016.880,48.455,388.690,166.367,55.360,160.066
C06283=1016.874,48.205,388.706,166.364,55.367,160.067
C06284=1016.869,47.956,388.721,166.361,55.376,160.068
C06285=1016.864,47.707,388.736,166.359,55.384,160.069
C06286=1016.859,47.457,388.750,166.357,55.392,160.070
C06287=1016.853,47.207,388.766,166.353,55.401,160.071
C06288=1016.848,46.957,388.781,166.351,55.408,160.072
C06289=1016.843,46.708,388.796,166.349,55.416,160.073
C06290=1016.838,46.459,388.811,166.347,55.424,160.074
C06291=1016.833,46.210,388.827,166.343,55.433,160.075
C06292=1016.828,45.960,388.842,166.341,55.441,160.076
C06293=1016.823,45.710,388.857,166.339,55.449,160.077
C06294=1016.817,45.461,388.873,166.337,55.457,160.078
C06295=1016.812,45.212,388.888,166.333,55.466,160.079
C06296=1016.807,44.963,388.903,166.331,55.474,160.080
C06297=1016.802,44.713,388.918,166.329,55.481,160.081
C06298=1016.797,44.463,388.933,166.325,55.490,160.082
C06299=1016.792,44.213,388.948,166.323,55.498,160.083
C06300=1016.787,43.964,388.963,166.321,55.506,160.084
C06301=1016.782,43.715,388.978,166.319,55.514,160.085
C06302=1016.776,43.465,388.994,166.315,55.522,160.086
C06303=1016.771,43.216,389.009,166.313,55.531,160.087
C06304=1016.766,42.934,389.026,166.310,55.539,160.088
C06305=1016.760,42.652,389.043,166.308,55.548,160.089
C06306=1016.754,42.370,389.060,166.305,55.558,160.090
C06307=1016.749,42.088,389.077,166.302,55.566,160.091
C06308=1016.744,41.839,389.092,166.300,55.575,160.093
C06309=1016.738,41.588,389.107,166.297,55.583,160.093
C06310=1016.733,41.339,389.122,166.294,55.591,160.095
C06311=1016.728,41.090,389.137,166.292,55.600,160.096
C06312=1016.723,40.840,389.151,166.289,55.608,160.097
C06313=1016.717,40.591,389.166,166.287,55.616,160.097
C06314=1016.712,40.342,389.181,166.285,55.624,160.099
C06315=1016.707,40.092,389.196,166.281,55.633,160.099
C06316=1016.702,39.842,389.211,166.279,55.641,160.101
C06317=1016.696,39.593,389.226,166.277,55.649,160.102
C06318=1016.691,39.343,389.240,166.274,55.658,160.103
C06319=1016.686,39.094,389.255,166.271,55.665,160.103
C06320=1016.681,38.844,389.269,166.269,55.673,160.105
C06321=1016.676,38.595,389.284,166.266,55.682,160.106
C06322=1016.671,38.346,389.300,166.264,55.690,160.107
C06323=1016.666,38.096,389.314,166.262,55.698,160.107
C06324=1016.660,37.847,389.329,166.258,55.706,160.108
C06325=1016.655,37.596,389.343,166.256,55.715,160.110
C06326=1016.650,37.347,389.359,166.254,55.723,160.111
C06327=1016.645,37.097,389.373,166.251,55.731,160.111
C06328=1016.639,36.848,389.388,166.249,55.739,160.112
C06329=1016.634,36.599,389.403,166.247,55.747,160.114
C06330=1016.629,36.349,389.417,166.243,55.756,160.114
C06331=1016.624,36.100,389.431,166.241,55.763,160.115
C06332=1016.619,35.850,389.446,166.239,55.772,160.116
C06333=1016.613,35.601,389.460,166.236,55.780,160.117
C06334=1016.608,35.351,389.475,166.234,55.788,160.118
C06335=1016.602,35.101,389.490,166.231,55.797,160.119
C06336=1016.597,34.851,389.504,166.229,55.805,160.121
C06337=1016.592,34.602,389.519,166.226,55.814,160.122
C06338=1016.587,34.352,389.533,166.223,55.822,160.122
C06339=1016.581,34.103,389.548,166.221,55.830,160.123
C06340=1016.576,33.854,389.562,166.218,55.838,160.124
C06341=1016.571,33.604,389.576,166.216,55.847,160.125
C06342=1016.566,33.355,389.591,166.214,55.855,160.127
C06343=1016.560,33.105,389.605,166.210,55.863,160.127
C06344=1016.556,32.855,389.620,166.208,55.871,160.128
C06345=1016.550,32.606,389.634,166.206,55.879,160.129
C06346=1016.545,32.356,389.649,166.203,55.888,160.130
C06347=1016.540,32.107,389.662,166.201,55.896,160.132
C06348=1016.535,31.858,389.678,166.198,55.904,160.132
C06349=1016.529,31.608,389.691,166.195,55.912,160.133
C06350=1016.524,31.358,389.705,166.193,55.921,160.134
C06351=1016.519,31.109,389.721,166.190,55.929,160.135
C06352=1016.513,30.860,389.734,166.187,55.937,160.136
C06353=1016.508,30.610,389.749,166.185,55.945,160.137
C06354=1016.503,30.361,389.763,166.182,55.954,160.138
C06355=1016.498,30.111,389.778,166.180,55.961,160.139
C06356=1016.492,29.861,389.792,166.178,55.970,160.140
C06357=1016.487,29.612,389.807,166.175,55.978,160.141
C06358=1016.482,29.362,389.821,166.172,55.986,160.142
C06359=1016.477,29.113,389.835,166.170,55.994,160.143
C06360=1016.472,28.863,389.849,166.167,56.003,160.144
C06361=1016.467,28.614,389.864,166.165,56.010,160.145
C06362=1016.461,28.364,389.878,166.163,56.019,160.146
C06363=1016.456,28.114,389.893,166.161,56.027,160.147
C06364=1016.451,27.865,389.906,166.157,56.035,160.148
C06365=1016.446,27.615,389.921,166.155,56.043,160.149
C06366=1016.440,27.366,389.936,166.153,56.051,160.150
C06367=1016.435,27.116,389.949,166.149,56.059,160.151
C06368=1016.429,26.834,389.965,166.147,56.069,160.152
C06369=1016.424,26.552,389.982,166.144,56.078,160.153
C06370=1016.418,26.270,389.998,166.142,56.088,160.154
C06371=1016.412,25.988,390.013,166.138,56.097,160.155
C06372=1016.407,25.739,390.027,166.136,56.105,160.156
C06373=1016.402,25.490,390.041,166.134,56.113,160.157
C06374=1016.397,25.241,390.056,166.130,56.121,160.158
C06375=1016.391,24.991,390.070,166.128,56.130,160.159
C06376=1016.386,24.742,390.083,166.125,56.138,160.160
C06377=1016.380,24.492,390.097,166.123,56.147,160.161
C06378=1016.375,24.242,390.111,166.121,56.154,160.162
C06379=1016.370,23.992,390.126,166.118,56.163,160.163
C06380=1016.364,23.743,390.139,166.116,56.171,160.164
C06381=1016.359,23.493,390.153,166.113,56.179,160.165
C06382=1016.354,23.244,390.167,166.110,56.187,160.166
C06383=1016.349,22.995,390.181,166.108,56.196,160.167
C06384=1016.344,22.745,390.195,166.106,56.203,160.168
C06385=1016.338,22.495,390.209,166.103,56.212,160.169
C06386=1016.333,22.246,390.223,166.101,56.220,160.170
C06387=1016.327,21.996,390.237,166.097,56.228,160.171
C06388=1016.323,21.746,390.251,166.095,56.237,160.172
C06389=1016.318,21.498,390.265,166.093,56.244,160.173
C06390=1016.312,21.248,390.279,166.090,56.253,160.174
C06391=1016.307,20.998,390.292,166.088,56.261,160.175
C06392=1016.302,20.748,390.307,166.085,56.269,160.176
C06393=1016.297,20.498,390.320,166.082,56.277,160.177
C06394=1016.291,20.249,390.334,166.080,56.285,160.177
C06395=1016.287,20.000,390.347,166.078,56.293,160.179
C06396=1016.281,19.750,390.361,166.075,56.302,160.180
C06397=1016.276,19.500,390.376,166.072,56.310,160.180
C06398=1016.271,19.251,390.390,166.070,56.318,160.182
C06399=1016.265,19.001,390.403,166.067,56.326,160.182
C06400=1016.260,18.752,390.417,166.065,56.334,160.183
C06401=1016.255,18.503,390.431,166.062,56.342,160.184
C06402=1016.250,18.253,390.445,166.059,56.351,160.185
C06403=1016.244,18.003,390.458,166.057,56.359,160.186
C06404=1016.239,17.753,390.472,166.055,56.366,160.187
C06405=1016.233,17.504,390.486,166.052,56.375,160.188
C06406=1016.229,17.255,390.500,166.050,56.383,160.189
C06407=1016.224,17.005,390.514,166.046,56.391,160.190
C06408=1016.219,16.755,390.527,166.044,56.400,160.191
C06409=1016.213,16.505,390.541,166.042,56.407,160.192
C06410=1016.208,16.256,390.554,166.039,56.416,160.193
C06411=1016.203,16.007,390.568,166.037,56.424,160.194
C06412=1016.198,15.757,390.581,166.035,56.432,160.195
C06413=1016.192,15.507,390.595,166.031,56.440,160.195
C06414=1016.187,15.258,390.608,166.029,56.448,160.197
C06415=1016.182,15.009,390.622,166.027,56.457,160.198
C06416=1016.177,14.758,390.635,166.024,56.465,160.198
C06417=1016.171,14.509,390.649,166.022,56.473,160.200
C06418=1016.166,14.260,390.663,166.019,56.481,160.200
C06419=1016.161,14.010,390.677,166.016,56.489,160.201
C06420=1016.156,13.760,390.690,166.014,56.497,160.202
C06421=1016.150,13.511,390.704,166.011,56.505,160.203
C06422=1016.146,13.261,390.717,166.008,56.513,160.204
C06423=1016.141,13.011,390.731,166.006,56.521,160.205
C06424=1016.135,12.762,390.744,166.004,56.529,160.206
C06425=1016.130,12.512,390.757,166.001,56.538,160.207
C06426=1016.125,12.263,390.771,165.999,56.546,160.208
C06427=1016.119,12.013,390.784,165.996,56.554,160.209
C06428=1016.113,11.763,390.797,165.994,56.563,160.210
C06429=1016.109,11.514,390.810,165.990,56.571,160.211
C06430=1016.103,11.264,390.824,165.988,56.579,160.212
C06431=1016.098,11.014,390.837,165.987,56.588,160.213
C06432=1016.092,10.735,390.852,165.983,56.597,160.214
C06433=1016.086,10.454,390.867,165.980,56.606,160.215
C06434=1016.080,10.173,390.882,165.977,56.615,160.216
C06435=1016.075,9.893,390.896,165.975,56.624,160.217
C06436=1016.068,9.644,390.910,165.971,56.632,160.218
C06437=1016.064,9.394,390.922,165.969,56.641,160.219
C06438=1016.058,9.144,390.936,165.966,56.649,160.220
C06439=1016.053,8.894,390.949,165.964,56.657,160.221
C06440=1016.048,8.646,390.962,165.962,56.665,160.222
C06441=1016.042,8.396,390.975,165.959,56.674,160.223
C06442=1016.037,8.146,390.989,165.956,56.681,160.223
C06443=1016.032,7.896,391.002,165.954,56.690,160.225
C06444=1016.026,7.647,391.015,165.951,56.698,160.225
C06445=1016.021,7.397,391.029,165.949,56.706,160.226
C06446=1016.016,7.147,391.041,165.946,56.714,160.227
C06447=1016.011,6.898,391.055,165.944,56.722,160.228
C06448=1016.006,6.649,391.067,165.941,56.730,160.229
C06449=1016.000,6.399,391.081,165.938,56.739,160.230
C06450=1015.995,6.149,391.094,165.936,56.747,160.231
C06451=1015.990,5.899,391.107,165.934,56.755,160.232
C06452=1015.985,5.650,391.121,165.931,56.763,160.233
C06453=1015.980,5.401,391.133,165.928,56.771,160.234
C06454=1015.974,5.151,391.146,165.926,56.779,160.235
C06455=1015.969,4.901,391.160,165.923,56.787,160.235
C06456=1015.964,4.651,391.173,165.921,56.795,160.237
C06457=1015.958,4.402,391.186,165.919,56.803,160.237
C06458=1015.954,4.153,391.199,165.915,56.811,160.238
C06459=1015.948,3.903,391.212,165.913,56.819,160.239
C06460=1015.944,3.653,391.225,165.911,56.827,160.240
C06461=1015.938,3.404,391.238,165.907,56.835,160.241
C06462=1015.933,3.154,391.251,165.906,56.844,160.242
C06463=1015.928,2.904,391.264,165.903,56.851,160.243
C06464=1015.922,2.654,391.278,165.900,56.859,160.244
C06465=1015.917,2.405,391.290,165.898,56.868,160.245
C06466=1015.912,2.155,391.303,165.896,56.875,160.246
C06467=1015.907,1.906,391.317,165.892,56.883,160.246
C06468=1015.902,1.656,391.330,165.890,56.892,160.247
C06469=1015.897,1.407,391.342,165.888,56.899,160.248
C06470=1015.891,1.157,391.355,165.884,56.908,160.249
C06471=1015.887,0.908,391.369,165.882,56.915,160.250
C06472=1015.881,0.658,391.382,165.880,56.924,160.251
C06473=1015.876,0.408,391.394,165.878,56.931,160.252
C06474=1015.871,0.158,391.407,165.874,56.939,160.252
C06475=1015.866,-0.091,391.421,165.872,56.947,160.253
C06476=1015.861,-0.341,391.434,165.870,56.955,160.255
C06477=1015.856,-0.590,391.446,165.868,56.963,160.255
C06478=1015.850,-0.840,391.459,165.864,56.971,160.256
C06479=1015.846,-1.090,391.472,165.862,56.979,160.257
C06480=1015.840,-1.339,391.486,165.860,56.986,160.258
C06481=1015.835,-1.588,391.498,165.858,56.995,160.259
C06482=1015.830,-1.838,391.511,165.854,57.003,160.260
C06483=1015.825,-2.088,391.524,165.852,57.011,160.261
C06484=1015.820,-2.337,391.536,165.850,57.018,160.261
C06485=1015.814,-2.587,391.550,165.847,57.026,160.262
C06486=1015.810,-2.836,391.563,165.844,57.034,160.263
C06487=1015.805,-3.087,391.576,165.841,57.042,160.264
C06488=1015.799,-3.336,391.588,165.839,57.049,160.265
C06489=1015.794,-3.586,391.601,165.837,57.058,160.266
C06490=1015.790,-3.835,391.614,165.834,57.066,160.267
C06491=1015.785,-4.084,391.628,165.831,57.074,160.267
C06492=1015.779,-4.334,391.640,165.829,57.081,160.268
C06493=1015.774,-4.584,391.653,165.827,57.089,160.269
C06494=1015.768,-4.834,391.666,165.823,57.097,160.270
C06495=1015.764,-5.084,391.678,165.821,57.105,160.271
C06496=1015.758,-5.368,391.693,165.819,57.114,160.272
C06497=1015.752,-5.653,391.706,165.815,57.124,160.273
C06498=1015.746,-5.938,391.721,165.812,57.133,160.274
C06499=1015.740,-6.222,391.735,165.810,57.142,160.275
C06500=1015.734,-6.472,391.748,165.807,57.150,160.276
C06501=1015.729,-6.722,391.760,165.804,57.159,160.277
C06502=1015.724,-6.971,391.773,165.802,57.166,160.278
C06503=1015.719,-7.222,391.785,165.799,57.174,160.278
C06504=1015.713,-7.471,391.797,165.796,57.182,160.279
C06505=1015.709,-7.720,391.810,165.795,57.190,160.280
C06506=1015.703,-7.970,391.822,165.791,57.199,160.281
C06507=1015.698,-8.220,391.835,165.789,57.206,160.282
C06508=1015.693,-8.469,391.847,165.786,57.214,160.283
C06509=1015.687,-8.719,391.860,165.783,57.222,160.283
C06510=1015.683,-8.969,391.872,165.781,57.230,160.285
C06511=1015.678,-9.218,391.884,165.779,57.238,160.286
C06512=1015.672,-9.468,391.896,165.776,57.246,160.286
C06513=1015.667,-9.717,391.909,165.773,57.254,160.287
C06514=1015.662,-9.966,391.921,165.771,57.262,160.288
C06515=1015.656,-10.217,391.933,165.769,57.269,160.289
C06516=1015.652,-10.466,391.946,165.765,57.278,160.289
C06517=1015.646,-10.716,391.958,165.763,57.286,160.291
C06518=1015.641,-10.966,391.971,165.761,57.294,160.292
C06519=1015.636,-11.215,391.984,165.758,57.302,160.292
C06520=1015.631,-11.465,391.995,165.755,57.310,160.293
C06521=1015.626,-11.715,392.008,165.753,57.317,160.294
C06522=1015.620,-11.964,392.020,165.751,57.325,160.295
C06523=1015.615,-12.213,392.033,165.747,57.333,160.296
C06524=1015.611,-12.464,392.045,165.745,57.341,160.296
C06525=1015.605,-12.713,392.057,165.743,57.348,160.297
C06526=1015.600,-12.963,392.069,165.739,57.357,160.298
C06527=1015.595,-13.212,392.082,165.737,57.364,160.299
C06528=1015.590,-13.462,392.094,165.735,57.372,160.300
C06529=1015.584,-13.712,392.106,165.732,57.380,160.301
C06530=1015.580,-13.961,392.119,165.729,57.388,160.301
C06531=1015.575,-14.211,392.130,165.727,57.396,160.302
C06532=1015.570,-14.461,392.143,165.724,57.403,160.303
C06533=1015.564,-14.710,392.156,165.722,57.411,160.304
C06534=1015.559,-14.960,392.167,165.720,57.419,160.305
C06535=1015.555,-15.210,392.180,165.716,57.427,160.305
C06536=1015.549,-15.459,392.192,165.714,57.435,160.306
C06537=1015.544,-15.709,392.204,165.712,57.442,160.307
C06538=1015.539,-15.959,392.217,165.710,57.450,160.308
C06539=1015.534,-16.208,392.229,165.706,57.458,160.309
C06540=1015.529,-16.458,392.240,165.704,57.466,160.310
C06541=1015.523,-16.708,392.253,165.702,57.474,160.311
C06542=1015.518,-16.958,392.264,165.698,57.482,160.311
C06543=1015.513,-17.207,392.277,165.696,57.490,160.312
C06544=1015.508,-17.457,392.288,165.694,57.497,160.313
C06545=1015.503,-17.706,392.300,165.690,57.505,160.314
C06546=1015.497,-17.957,392.313,165.689,57.514,160.315
C06547=1015.492,-18.206,392.324,165.686,57.522,160.316
C06548=1015.487,-18.456,392.336,165.683,57.530,160.316
C06549=1015.482,-18.705,392.348,165.681,57.538,160.317
C06550=1015.477,-18.955,392.360,165.678,57.545,160.318
C06551=1015.472,-19.204,392.372,165.676,57.553,160.319
C06552=1015.467,-19.451,392.383,165.673,57.561,160.320
C06553=1015.461,-19.697,392.395,165.670,57.568,160.320
C06554=1015.456,-19.944,392.407,165.668,57.576,160.321
C06555=1015.451,-20.190,392.418,165.665,57.584,160.322
C06556=1015.446,-20.436,392.430,165.663,57.591,160.323
C06557=1015.441,-20.683,392.442,165.660,57.600,160.324
C06558=1015.436,-20.930,392.454,165.657,57.607,160.325
C06559=1015.431,-21.175,392.466,165.655,57.615,160.325
C06560=1015.425,-21.452,392.478,165.652,57.623,160.326
C06561=1015.420,-21.729,392.492,165.649,57.632,160.327
C06562=1015.414,-22.005,392.505,165.646,57.641,160.328
C06563=1015.408,-22.282,392.517,165.643,57.649,160.329
C06564=1015.404,-22.532,392.529,165.641,57.657,160.330
C06565=1015.398,-22.781,392.541,165.639,57.665,160.331
C06566=1015.393,-23.031,392.553,165.636,57.673,160.331
C06567=1015.388,-23.281,392.565,165.633,57.681,160.332
C06568=1015.382,-23.530,392.577,165.631,57.688,160.333
C06569=1015.377,-23.780,392.588,165.628,57.695,160.334
C06570=1015.372,-24.030,392.600,165.626,57.703,160.334
C06571=1015.367,-24.279,392.612,165.623,57.711,160.335
C06572=1015.362,-24.529,392.624,165.620,57.719,160.336
C06573=1015.357,-24.779,392.635,165.618,57.727,160.337
C06574=1015.352,-25.028,392.647,165.615,57.734,160.337
C06575=1015.347,-25.278,392.659,165.613,57.742,160.338
C06576=1015.342,-25.528,392.670,165.610,57.749,160.339
C06577=1015.337,-25.777,392.682,165.607,57.758,160.340
C06578=1015.331,-26.027,392.694,165.604,57.765,160.341
C06579=1015.326,-26.276,392.705,165.602,57.772,160.341
C06580=1015.321,-26.526,392.717,165.600,57.780,160.342
C06581=1015.317,-26.776,392.729,165.598,57.788,160.343
C06582=1015.312,-27.025,392.741,165.595,57.795,160.344
C06583=1015.307,-27.275,392.753,165.591,57.803,160.344
C06584=1015.302,-27.525,392.764,165.589,57.811,160.345
C06585=1015.297,-27.775,392.775,165.586,57.818,160.346
C06586=1015.292,-28.025,392.787,165.584,57.826,160.347
C06587=1015.286,-28.274,392.798,165.582,57.834,160.348
C06588=1015.281,-28.524,392.809,165.579,57.842,160.348
C06589=1015.276,-28.773,392.821,165.576,57.850,160.349
C06590=1015.271,-29.023,392.833,165.573,57.857,160.350
C06591=1015.266,-29.273,392.844,165.570,57.865,160.351
C06592=1015.260,-29.522,392.855,165.568,57.873,160.351
C06593=1015.255,-29.772,392.867,165.566,57.880,160.352
C06594=1015.250,-30.022,392.878,165.564,57.888,160.353
C06595=1015.245,-30.272,392.890,165.560,57.896,160.354
C06596=1015.239,-30.521,392.901,165.557,57.903,160.355
C06597=1015.234,-30.771,392.912,165.555,57.911,160.355
C06598=1015.229,-31.021,392.924,165.553,57.919,160.356
C06599=1015.224,-31.270,392.935,165.551,57.927,160.357
C06600=1015.219,-31.520,392.946,165.547,57.934,160.358
C06601=1015.214,-31.770,392.957,165.545,57.942,160.358
C06602=1015.209,-32.020,392.969,165.542,57.950,160.359
C06603=1015.204,-32.269,392.979,165.540,57.957,160.360
C06604=1015.199,-32.519,392.991,165.536,57.965,160.361
C06605=1015.194,-32.769,393.002,165.534,57.973,160.362
C06606=1015.189,-33.018,393.013,165.532,57.981,160.362
C06607=1015.184,-33.268,393.025,165.529,57.988,160.363
C06608=1015.179,-33.518,393.036,165.527,57.995,160.364
C06609=1015.173,-33.767,393.047,165.524,58.003,160.364
C06610=1015.168,-34.017,393.058,165.521,58.011,160.365
C06611=1015.163,-34.267,393.070,165.519,58.019,160.366
C06612=1015.159,-34.516,393.081,165.516,58.026,160.367
C06613=1015.153,-34.766,393.092,165.514,58.033,160.368
C06614=1015.148,-35.015,393.103,165.511,58.041,160.368
C06615=1015.143,-35.266,393.114,165.509,58.048,160.369
C06616=1015.138,-35.516,393.126,165.505,58.056,160.370
C06617=1015.132,-35.765,393.136,165.503,58.064,160.370
C06618=1015.127,-36.015,393.148,165.500,58.071,160.371
C06619=1015.123,-36.264,393.159,165.498,58.078,160.372
C06620=1015.118,-36.514,393.170,165.495,58.086,160.373
C06621=1015.112,-36.763,393.181,165.493,58.093,160.373
C06622=1015.108,-37.014,393.192,165.490,58.101,160.374
C06623=1015.103,-37.264,393.204,165.488,58.108,160.375
C06624=1015.097,-37.538,393.216,165.485,58.117,160.376
C06625=1015.091,-37.813,393.228,165.482,58.125,160.376
C06626=1015.087,-38.090,393.240,165.478,58.134,160.377
C06627=1015.081,-38.365,393.253,165.476,58.141,160.378
C06628=1015.075,-38.614,393.264,165.473,58.148,160.379
C06629=1015.070,-38.865,393.275,165.471,58.156,160.379
C06630=1015.066,-39.114,393.286,165.467,58.164,160.380
C06631=1015.061,-39.364,393.297,165.465,58.172,160.381
C06632=1015.055,-39.613,393.308,165.462,58.179,160.381
C06633=1015.050,-39.864,393.319,165.460,58.186,160.382
C06634=1015.045,-40.112,393.329,165.458,58.194,160.383
C06635=1015.041,-40.363,393.340,165.455,58.201,160.384
C06636=1015.035,-40.612,393.351,165.453,58.208,160.384
C06637=1015.030,-40.862,393.362,165.449,58.217,160.385
C06638=1015.025,-41.112,393.372,165.447,58.225,160.386
C06639=1015.020,-41.361,393.384,165.444,58.232,160.386
C06640=1015.015,-41.611,393.394,165.442,58.239,160.387
C06641=1015.010,-41.861,393.405,165.439,58.247,160.388
C06642=1015.005,-42.111,393.415,165.437,58.254,160.389
C06643=1015.000,-42.360,393.427,165.433,58.262,160.389
C06644=1014.994,-42.610,393.437,165.431,58.270,160.390
C06645=1014.989,-42.860,393.448,165.429,58.277,160.391
C06646=1014.984,-43.109,393.459,165.426,58.284,160.391
C06647=1014.980,-43.360,393.469,165.424,58.292,160.392
C06648=1014.974,-43.609,393.480,165.421,58.299,160.393
C06649=1014.970,-43.859,393.491,165.419,58.307,160.394
C06650=1014.964,-44.108,393.502,165.416,58.314,160.394
C06651=1014.959,-44.358,393.512,165.414,58.322,160.395
C06652=1014.954,-44.607,393.523,165.410,58.329,160.396
C06653=1014.949,-44.858,393.533,165.407,58.336,160.396
C06654=1014.944,-45.107,393.545,165.405,58.344,160.397
C06655=1014.939,-45.357,393.554,165.402,58.351,160.398
C06656=1014.934,-45.607,393.566,165.400,58.358,160.398
C06657=1014.928,-45.857,393.576,165.397,58.366,160.399
C06658=1014.924,-46.106,393.587,165.395,58.373,160.400
C06659=1014.919,-46.356,393.597,165.392,58.380,160.400
C06660=1014.914,-46.606,393.608,165.390,58.388,160.401
C06661=1014.909,-46.855,393.618,165.387,58.395,160.402
C06662=1014.904,-47.106,393.629,165.384,58.402,160.402
C06663=1014.899,-47.354,393.640,165.382,58.410,160.403
C06664=1014.894,-47.605,393.650,165.379,58.417,160.404
C06665=1014.888,-47.854,393.661,165.377,58.424,160.404
C06666=1014.884,-48.104,393.672,165.374,58.431,160.405
C06667=1014.879,-48.354,393.682,165.372,58.439,160.406
C06668=1014.874,-48.603,393.692,165.369,58.446,160.407
C06669=1014.869,-48.853,393.703,165.366,58.453,160.407
C06670=1014.864,-49.103,393.713,165.363,58.461,160.408
C06671=1014.859,-49.352,393.724,165.361,58.468,160.408
C06672=1014.854,-49.603,393.735,165.359,58.475,160.409
C06673=1014.849,-49.852,393.746,165.356,58.483,160.410
C06674=1014.844,-50.102,393.756,165.353,58.490,160.410
C06675=1014.840,-50.352,393.766,165.350,58.497,160.411
C06676=1014.834,-50.602,393.776,165.348,58.504,160.412
C06677=1014.829,-50.851,393.788,165.345,58.511,160.412
C06678=1014.825,-51.101,393.798,165.342,58.518,160.413
C06679=1014.819,-51.351,393.808,165.340,58.526,160.414
C06680=1014.814,-51.600,393.818,165.337,58.533,160.414
C06681=1014.810,-51.851,393.828,165.335,58.541,160.415
C06682=1014.805,-52.100,393.838,165.331,58.549,160.415
C06683=1014.799,-52.350,393.848,165.329,58.556,160.416
C06684=1014.794,-52.599,393.859,165.327,58.563,160.417
C06685=1014.789,-52.849,393.869,165.324,58.571,160.418
C06686=1014.784,-53.099,393.879,165.321,58.578,160.418
C06687=1014.779,-53.349,393.889,165.319,58.586,160.419
C06688=1014.773,-53.625,393.899,165.316,58.594,160.420
C06689=1014.768,-53.900,393.911,165.313,58.602,160.420
C06690=1014.761,-54.176,393.922,165.311,58.610,160.421
C06691=1014.756,-54.452,393.933,165.307,58.618,160.422
C06692=1014.751,-54.702,393.943,165.305,58.625,160.423
C06693=1014.746,-54.952,393.953,165.302,58.633,160.423
C06694=1014.741,-55.201,393.963,165.299,58.640,160.424
C06695=1014.736,-55.451,393.973,165.296,58.647,160.424
C06696=1014.731,-55.701,393.983,165.294,58.655,160.425
C06697=1014.726,-55.950,393.993,165.291,58.662,160.426
C06698=1014.721,-56.200,394.003,165.288,58.669,160.426
C06699=1014.716,-56.450,394.012,165.285,58.677,160.427
C06700=1014.710,-56.700,394.023,165.282,58.684,160.427
C06701=1014.705,-56.949,394.032,165.280,58.692,160.428
C06702=1014.701,-57.198,394.042,165.278,58.699,160.429
C06703=1014.695,-57.449,394.052,165.275,58.706,160.430
C06704=1014.690,-57.698,394.062,165.272,58.713,160.430
C06705=1014.685,-57.948,394.072,165.270,58.720,160.431
C06706=1014.681,-58.198,394.083,165.267,58.727,160.431
C06707=1014.676,-58.447,394.093,165.264,58.734,160.432
C06708=1014.671,-58.698,394.102,165.261,58.742,160.432
C06709=1014.666,-58.947,394.112,165.259,58.749,160.433
C06710=1014.661,-59.197,394.122,165.257,58.757,160.434
C06711=1014.656,-59.447,394.132,165.254,58.764,160.435
C06712=1014.651,-59.696,394.142,165.251,58.771,160.435
C06713=1014.645,-59.946,394.152,165.249,58.778,160.436
C06714=1014.641,-60.196,394.161,165.247,58.785,160.437
C06715=1014.636,-60.445,394.171,165.244,58.792,160.437
C06716=1014.631,-60.696,394.181,165.242,58.799,160.438
C06717=1014.626,-60.945,394.191,165.239,58.806,160.438
C06718=1014.621,-61.195,394.200,165.236,58.813,160.439
C06719=1014.616,-61.445,394.210,165.233,58.820,160.439
C06720=1014.611,-61.694,394.220,165.231,58.828,160.440
C06721=1014.606,-61.944,394.230,165.228,58.835,160.441
C06722=1014.601,-62.194,394.240,165.225,58.841,160.441
C06723=1014.596,-62.444,394.249,165.222,58.848,160.442
C06724=1014.591,-62.693,394.259,165.219,58.855,160.442
C06725=1014.586,-62.943,394.269,165.218,58.862,160.443
C06726=1014.581,-63.193,394.279,165.215,58.869,160.444
C06727=1014.576,-63.443,394.288,165.212,58.876,160.444
C06728=1014.571,-63.692,394.298,165.210,58.884,160.445
C06729=1014.566,-63.942,394.308,165.207,58.891,160.445
C06730=1014.561,-64.192,394.318,165.204,58.897,160.446
C06731=1014.557,-64.442,394.327,165.201,58.904,160.446
C06732=1014.551,-64.692,394.337,165.199,58.911,160.447
C06733=1014.546,-64.941,394.347,165.197,58.918,160.448
C06734=1014.542,-65.191,394.357,165.194,58.925,160.448
C06735=1014.537,-65.441,394.366,165.191,58.932,160.448
C06736=1014.532,-65.691,394.376,165.188,58.939,160.449
C06737=1014.527,-65.940,394.386,165.186,58.946,160.450
C06738=1014.523,-66.191,394.395,165.184,58.953,160.450
C06739=1014.518,-66.440,394.405,165.180,58.959,160.451
C06740=1014.513,-66.689,394.415,165.178,58.966,160.451
C06741=1014.508,-66.939,394.425,165.175,58.973,160.452
C06742=1014.503,-67.189,394.434,165.173,58.979,160.452
C06743=1014.499,-67.439,394.444,165.170,58.987,160.453
C06744=1014.494,-67.688,394.454,165.168,58.994,160.453
C06745=1014.489,-67.938,394.463,165.164,59.000,160.454
C06746=1014.484,-68.188,394.473,165.163,59.007,160.455
C06747=1014.479,-68.438,394.482,165.160,59.014,160.455
C06748=1014.474,-68.688,394.492,165.157,59.021,160.455
C06749=1014.470,-68.937,394.502,165.154,59.028,160.456
C06750=1014.465,-69.187,394.511,165.152,59.034,160.457
C06751=1014.460,-69.437,394.521,165.149,59.041,160.457
C06752=1014.454,-69.714,394.532,165.146,59.048,160.458
C06753=1014.449,-69.991,394.542,165.143,59.056,160.458
C06754=1014.443,-70.267,394.553,165.141,59.064,160.459
C06755=1014.439,-70.544,394.563,165.138,59.071,160.460
C06756=1014.434,-70.794,394.573,165.135,59.077,160.460
C06757=1014.429,-71.044,394.582,165.132,59.084,160.460
C06758=1014.424,-71.293,394.592,165.130,59.090,160.461
C06759=1014.420,-71.543,394.601,165.127,59.097,160.461
C06760=1014.415,-71.793,394.611,165.125,59.103,160.462
C06761=1014.410,-72.042,394.621,165.122,59.111,160.463
C06762=1014.406,-72.292,394.630,165.119,59.117,160.463
C06763=1014.400,-72.542,394.640,165.117,59.124,160.464
C06764=1014.396,-72.792,394.649,165.114,59.130,160.464
C06765=1014.391,-73.042,394.659,165.111,59.137,160.464
C06766=1014.386,-73.292,394.668,165.109,59.143,160.465
C06767=1014.381,-73.541,394.677,165.106,59.150,160.465
///RCONF 1,0,0,0,1,0,0,0,0,0,0,0,0,0,0,0,0,0,0,0,0,0,0,0
C06768=1014.377,-73.791,394.687,165.104,59.157,160.466
C06769=1014.372,-74.041,394.696,165.101,59.163,160.466
C06770=1014.368,-74.291,394.705,165.098,59.169,160.467
C06771=1014.363,-74.540,394.715,165.096,59.176,160.467
C06772=1014.358,-74.790,394.724,165.093,59.183,160.468
C06773=1014.353,-75.040,394.733,165.091,59.189,160.468
C06774=1014.348,-75.289,394.743,165.088,59.196,160.469
C06775=1014.344,-75.539,394.752,165.085,59.203,160.469
C06776=1014.339,-75.789,394.761,165.082,59.209,160.470
C06777=1014.334,-76.039,394.769,165.081,59.216,160.470
C06778=1014.329,-76.288,394.779,165.077,59.223,160.471
C06779=1014.324,-76.538,394.788,165.075,59.230,160.471
C06780=1014.319,-76.788,394.797,165.072,59.236,160.472
C06781=1014.315,-77.038,394.806,165.070,59.243,160.472
C06782=1014.310,-77.287,394.815,165.067,59.249,160.473
C06783=1014.305,-77.537,394.824,165.065,59.256,160.473
C06784=1014.300,-77.787,394.833,165.062,59.263,160.474
C06785=1014.296,-78.037,394.842,165.060,59.269,160.474
C06786=1014.291,-78.287,394.852,165.057,59.276,160.475
C06787=1014.285,-78.536,394.860,165.054,59.282,160.475
C06788=1014.281,-78.786,394.869,165.052,59.289,160.476
C06789=1014.276,-79.036,394.879,165.049,59.295,160.476
C06790=1014.271,-79.286,394.887,165.046,59.302,160.476
C06791=1014.266,-79.536,394.897,165.044,59.309,160.477
C06792=1014.262,-79.786,394.906,165.041,59.315,160.477
C06793=1014.256,-80.035,394.914,165.039,59.321,160.478
C06794=1014.252,-80.285,394.923,165.036,59.328,160.479
C06795=1014.247,-80.535,394.933,165.034,59.334,160.479
C06796=1014.242,-80.785,394.941,165.030,59.341,160.479
C06797=1014.238,-81.035,394.950,165.028,59.348,160.480
C06798=1014.232,-81.285,394.959,165.026,59.354,160.480
C06799=1014.228,-81.535,394.968,165.023,59.361,160.481
C06800=1014.223,-81.785,394.976,165.020,59.368,160.481
C06801=1014.217,-82.034,394.985,165.018,59.374,160.482
C06802=1014.213,-82.284,394.994,165.015,59.381,160.482
C06803=1014.208,-82.533,395.002,165.012,59.387,160.483
C06804=1014.204,-82.783,395.011,165.010,59.394,160.483
C06805=1014.198,-83.033,395.019,165.007,59.401,160.484
C06806=1014.193,-83.283,395.028,165.004,59.408,160.484
C06807=1014.189,-83.533,395.037,165.002,59.414,160.485
C06808=1014.184,-83.783,395.045,164.999,59.420,160.485
C06809=1014.179,-84.033,395.054,164.997,59.427,160.486
C06810=1014.174,-84.282,395.062,164.994,59.434,160.486
C06811=1014.170,-84.532,395.071,164.992,59.440,160.487
C06812=1014.165,-84.782,395.080,164.989,59.446,160.487
C06813=1014.159,-85.032,395.088,164.986,59.453,160.487
C06814=1014.155,-85.282,395.097,164.984,59.459,160.488
C06815=1014.150,-85.531,395.106,164.980,59.466,160.488
C06816=1014.145,-85.810,395.115,164.978,59.473,160.489
C06817=1014.139,-86.089,395.125,164.975,59.480,160.489
C06818=1014.134,-86.368,395.133,164.973,59.487,160.490
C06819=1014.129,-86.646,395.143,164.969,59.494,160.490
C06820=1014.123,-86.896,395.152,164.967,59.501,160.491
C06821=1014.119,-87.145,395.161,164.965,59.507,160.491
C06822=1014.114,-87.395,395.169,164.961,59.514,160.491
C06823=1014.110,-87.646,395.178,164.959,59.520,160.492
C06824=1014.105,-87.895,395.186,164.956,59.526,160.492
C06825=1014.099,-88.145,395.194,164.954,59.532,160.493
C06826=1014.095,-88.394,395.203,164.951,59.539,160.493
C06827=1014.090,-88.644,395.212,164.948,59.545,160.493
C06828=1014.086,-88.895,395.220,164.946,59.552,160.494
C06829=1014.081,-89.144,395.229,164.944,59.558,160.495
C06830=1014.076,-89.393,395.237,164.941,59.564,160.495
C06831=1014.071,-89.644,395.246,164.938,59.570,160.495
C06832=1014.067,-89.894,395.253,164.936,59.576,160.496
C06833=1014.062,-90.144,395.263,164.933,59.583,160.496
C06834=1014.057,-90.393,395.271,164.931,59.589,160.496
C06835=1014.052,-90.643,395.279,164.928,59.595,160.497
C06836=1014.048,-90.893,395.288,164.925,59.601,160.497
C06837=1014.043,-91.142,395.296,164.923,59.607,160.498
C06838=1014.039,-91.392,395.305,164.920,59.614,160.498
C06839=1014.034,-91.643,395.313,164.918,59.620,160.498
C06840=1014.029,-91.892,395.321,164.915,59.626,160.499
C06841=1014.025,-92.142,395.330,164.912,59.632,160.499
C06842=1014.020,-92.392,395.337,164.909,59.638,160.499
C06843=1014.016,-92.641,395.346,164.907,59.644,160.500
C06844=1014.010,-92.891,395.355,164.904,59.650,160.500
C06845=1014.005,-93.141,395.362,164.902,59.656,160.501
C06846=1014.001,-93.391,395.371,164.900,59.662,160.501
C06847=1013.996,-93.640,395.380,164.898,59.668,160.502
C06848=1013.992,-93.891,395.388,164.894,59.674,160.501
C06849=1013.987,-94.140,395.396,164.891,59.680,160.502
C06850=1013.982,-94.390,395.405,164.889,59.686,160.502
C06851=1013.978,-94.640,395.413,164.886,59.693,160.503
C06852=1013.973,-94.889,395.421,164.884,59.699,160.503
C06853=1013.969,-95.139,395.430,164.881,59.704,160.503
C06854=1013.964,-95.390,395.438,164.879,59.710,160.504
C06855=1013.959,-95.639,395.446,164.877,59.716,160.504
C06856=1013.955,-95.889,395.454,164.874,59.723,160.505
C06857=1013.950,-96.138,395.463,164.871,59.728,160.505
C06858=1013.945,-96.389,395.470,164.869,59.734,160.505
C06859=1013.941,-96.639,395.479,164.866,59.740,160.506
C06860=1013.936,-96.888,395.488,164.864,59.745,160.506
C06861=1013.932,-97.139,395.496,164.860,59.752,160.506
C06862=1013.927,-97.388,395.504,164.858,59.758,160.507
C06863=1013.922,-97.638,395.512,164.855,59.763,160.507
C06864=1013.918,-97.887,395.520,164.853,59.769,160.507
C06865=1013.913,-98.138,395.528,164.851,59.775,160.508
C06866=1013.908,-98.387,395.537,164.847,59.781,160.508
C06867=1013.904,-98.637,395.544,164.845,59.787,160.508
C06868=1013.899,-98.887,395.552,164.843,59.793,160.509
C06869=1013.895,-99.137,395.561,164.841,59.799,160.509
C06870=1013.890,-99.387,395.568,164.837,59.805,160.509
C06871=1013.885,-99.636,395.576,164.835,59.811,160.509
C06872=1013.880,-99.886,395.584,164.833,59.817,160.510
C06873=1013.876,-100.136,395.592,164.831,59.823,160.510
C06874=1013.871,-100.386,395.599,164.828,59.828,160.511
C06875=1013.866,-100.635,395.608,164.825,59.835,160.511
C06876=1013.861,-100.886,395.615,164.822,59.841,160.511
C06877=1013.857,-101.135,395.623,164.820,59.846,160.511
C06878=1013.852,-101.386,395.631,164.817,59.852,160.512
C06879=1013.848,-101.635,395.639,164.815,59.858,160.512
C06880=1013.843,-101.916,395.647,164.812,59.865,160.513
C06881=1013.838,-102.196,395.656,164.809,59.871,160.513
C06882=1013.832,-102.478,395.666,164.806,59.878,160.513
C06883=1013.827,-102.758,395.675,164.804,59.884,160.514
C06884=1013.823,-103.008,395.682,164.800,59.890,160.514
C06885=1013.818,-103.258,395.690,164.798,59.896,160.514
C06886=1013.813,-103.507,395.698,164.795,59.902,160.515
C06887=1013.809,-103.757,395.705,164.793,59.907,160.515
C06888=1013.804,-104.007,395.713,164.790,59.913,160.515
C06889=1013.799,-104.257,395.720,164.788,59.918,160.515
C06890=1013.794,-104.507,395.728,164.786,59.924,160.516
C06891=1013.790,-104.756,395.736,164.783,59.930,160.516
C06892=1013.785,-105.006,395.744,164.781,59.936,160.516
C06893=1013.780,-105.256,395.751,164.778,59.941,160.517
C06894=1013.776,-105.505,395.759,164.776,59.947,160.517
C06895=1013.772,-105.756,395.767,164.773,59.952,160.517
C06896=1013.767,-106.006,395.775,164.771,59.959,160.518
C06897=1013.762,-106.256,395.782,164.768,59.964,160.518
C06898=1013.758,-106.505,395.791,164.766,59.970,160.518
C06899=1013.753,-106.755,395.798,164.763,59.975,160.518
C06900=1013.748,-107.005,395.806,164.760,59.981,160.519
C06901=1013.744,-107.255,395.813,164.758,59.987,160.519
C06902=1013.740,-107.504,395.820,164.755,59.992,160.519
C06903=1013.735,-107.755,395.828,164.753,59.997,160.519
C06904=1013.730,-108.004,395.836,164.750,60.003,160.520
C06905=1013.726,-108.254,395.843,164.748,60.009,160.520
C06906=1013.721,-108.504,395.851,164.746,60.015,160.521
C06907=1013.716,-108.754,395.858,164.743,60.020,160.521
C06908=1013.712,-109.003,395.865,164.740,60.025,160.521
C06909=1013.707,-109.254,395.873,164.738,60.031,160.521
C06910=1013.702,-109.503,395.880,164.735,60.037,160.521
C06911=1013.698,-109.753,395.888,164.733,60.043,160.522
C06912=1013.693,-110.003,395.895,164.730,60.048,160.522
C06913=1013.689,-110.253,395.903,164.727,60.053,160.522
C06914=1013.684,-110.502,395.910,164.725,60.059,160.522
C06915=1013.680,-110.752,395.918,164.722,60.065,160.523
C06916=1013.674,-111.002,395.925,164.720,60.070,160.523
C06917=1013.670,-111.252,395.932,164.717,60.075,160.523
C06918=1013.666,-111.502,395.939,164.715,60.081,160.524
C06919=1013.661,-111.752,395.947,164.712,60.087,160.524
C06920=1013.656,-112.002,395.954,164.709,60.092,160.524
C06921=1013.652,-112.252,395.961,164.706,60.097,160.524
C06922=1013.648,-112.501,395.969,164.705,60.102,160.524
C06923=1013.643,-112.752,395.977,164.703,60.108,160.525
C06924=1013.638,-113.001,395.984,164.700,60.114,160.525
C06925=1013.633,-113.251,395.991,164.697,60.119,160.525
C06926=1013.629,-113.501,395.998,164.694,60.124,160.525
C06927=1013.624,-113.751,396.005,164.692,60.130,160.525
C06928=1013.620,-114.001,396.013,164.690,60.135,160.526
C06929=1013.616,-114.250,396.020,164.687,60.140,160.526
C06930=1013.611,-114.500,396.027,164.685,60.146,160.526
C06931=1013.607,-114.750,396.035,164.682,60.151,160.527
C06932=1013.602,-115.001,396.042,164.679,60.157,160.527
C06933=1013.597,-115.250,396.049,164.678,60.161,160.527
C06934=1013.593,-115.500,396.056,164.675,60.167,160.527
C06935=1013.588,-115.749,396.064,164.672,60.172,160.527
C06936=1013.584,-115.999,396.070,164.669,60.177,160.528
C06937=1013.579,-116.249,396.077,164.667,60.183,160.528
C06938=1013.574,-116.499,396.085,164.665,60.188,160.528
C06939=1013.570,-116.749,396.092,164.662,60.193,160.528
C06940=1013.566,-116.999,396.099,164.659,60.198,160.528
C06941=1013.561,-117.248,396.106,164.657,60.204,160.528
C06942=1013.557,-117.499,396.112,164.655,60.208,160.529
C06943=1013.552,-117.748,396.120,164.652,60.214,160.529
C06944=1013.548,-118.029,396.128,164.650,60.220,160.529
C06945=1013.542,-118.310,396.136,164.646,60.226,160.529
C06946=1013.537,-118.591,396.144,164.644,60.232,160.530
C06947=1013.531,-118.872,396.151,164.641,60.237,160.530
C06948=1013.527,-119.121,396.159,164.639,60.242,160.530
C06949=1013.523,-119.372,396.165,164.636,60.248,160.530
C06950=1013.519,-119.621,396.173,164.634,60.253,160.531
C06951=1013.514,-119.871,396.179,164.631,60.258,160.531
C06952=1013.509,-120.122,396.187,164.629,60.263,160.531
C06953=1013.504,-120.371,396.194,164.627,60.268,160.531
C06954=1013.500,-120.621,396.200,164.624,60.274,160.531
C06955=1013.495,-120.871,396.208,164.621,60.279,160.532
C06956=1013.491,-121.121,396.214,164.620,60.284,160.532
C06957=1013.486,-121.370,396.221,164.616,60.288,160.532
C06958=1013.482,-121.621,396.228,164.615,60.293,160.532
C06959=1013.478,-121.870,396.235,164.612,60.299,160.532
C06960=1013.473,-122.120,396.241,164.609,60.304,160.532
C06961=1013.469,-122.370,396.249,164.607,60.309,160.533
C06962=1013.465,-122.620,396.255,164.604,60.313,160.533
C06963=1013.459,-122.869,396.262,164.602,60.318,160.533
C06964=1013.455,-123.120,396.269,164.599,60.324,160.533
C06965=1013.451,-123.369,396.276,164.598,60.328,160.533
C06966=1013.446,-123.619,396.282,164.594,60.333,160.533
C06967=1013.442,-123.869,396.290,164.592,60.338,160.533
C06968=1013.438,-124.119,396.297,164.590,60.343,160.534
C06969=1013.433,-124.369,396.303,164.587,60.349,160.534
C06970=1013.429,-124.619,396.310,164.585,60.353,160.534
C06971=1013.425,-124.869,396.317,164.582,60.358,160.534
C06972=1013.420,-125.118,396.324,164.580,60.363,160.534
C06973=1013.416,-125.369,396.330,164.577,60.368,160.534
C06974=1013.410,-125.618,396.337,164.575,60.372,160.535
C06975=1013.406,-125.868,396.344,164.572,60.378,160.535
C06976=1013.402,-126.118,396.350,164.571,60.383,160.535
C06977=1013.397,-126.368,396.357,164.567,60.387,160.535
C06978=1013.392,-126.618,396.363,164.566,60.392,160.535
C06979=1013.388,-126.868,396.370,164.562,60.397,160.535
C06980=1013.384,-127.118,396.376,164.561,60.402,160.535
C06981=1013.379,-127.368,396.383,164.559,60.406,160.536
C06982=1013.374,-127.617,396.390,164.555,60.411,160.536
C06983=1013.370,-127.868,396.396,164.554,60.416,160.536
C06984=1013.366,-128.116,396.403,164.550,60.421,160.536
C06985=1013.362,-128.366,396.410,164.549,60.425,160.536
C06986=1013.358,-128.616,396.417,164.546,60.430,160.536
C06987=1013.354,-128.866,396.425,164.544,60.434,160.536
C06988=1013.351,-129.115,396.433,164.542,60.437,160.536
C06989=1013.347,-129.364,396.442,164.538,60.439,160.535
C06990=1013.345,-129.614,396.452,164.537,60.442,160.536
C06991=1013.342,-129.864,396.463,164.535,60.444,160.535
C06992=1013.340,-130.114,396.473,164.533,60.445,160.535
C06993=1013.339,-130.363,396.486,164.529,60.446,160.534
C06994=1013.338,-130.613,396.498,164.528,60.447,160.534
C06995=1013.336,-130.863,396.510,164.526,60.448,160.533
C06996=1013.336,-131.112,396.524,164.524,60.446,160.532
C06997=1013.336,-131.362,396.538,164.522,60.446,160.532
C06998=1013.335,-131.612,396.552,164.519,60.445,160.531
C06999=1013.336,-131.861,396.567,164.518,60.444,160.530
C07000=1013.336,-132.111,396.584,164.516,60.441,160.529
C07001=1013.338,-132.361,396.599,164.514,60.439,160.528
C07002=1013.339,-132.610,396.617,164.511,60.436,160.526
C07003=1013.341,-132.860,396.634,164.509,60.433,160.525
C07004=1013.342,-133.110,396.653,164.508,60.429,160.524
C07005=1013.345,-133.359,396.672,164.505,60.425,160.522
C07006=1013.348,-133.609,396.691,164.504,60.420,160.521
C07007=1013.351,-133.858,396.711,164.501,60.415,160.519
C07008=1013.124,-133.884,396.290,164.486,60.704,160.568
C07009=1013.121,-133.635,396.270,164.489,60.708,160.570
C07010=1013.118,-133.386,396.250,164.490,60.713,160.571
C07011=1013.116,-133.136,396.232,164.492,60.717,160.573
C07012=1013.113,-132.886,396.214,164.494,60.720,160.574
C07013=1013.112,-132.637,396.196,164.496,60.724,160.575
C07014=1013.111,-132.387,396.180,164.498,60.726,160.576
C07015=1013.110,-132.137,396.162,164.500,60.728,160.577
C07016=1013.109,-131.887,396.147,164.502,60.731,160.578
C07017=1013.108,-131.637,396.132,164.505,60.732,160.579
C07018=1013.109,-131.388,396.117,164.506,60.733,160.580
C07019=1013.109,-131.139,396.103,164.508,60.734,160.581
C07020=1013.110,-130.889,396.090,164.510,60.735,160.582
C07021=1013.111,-130.639,396.076,164.512,60.734,160.582
C07022=1013.112,-130.389,396.065,164.515,60.733,160.583
C07023=1013.113,-130.139,396.053,164.518,60.733,160.584
C07024=1013.116,-129.890,396.042,164.519,60.731,160.584
C07025=1013.118,-129.640,396.032,164.521,60.730,160.585
C07026=1013.120,-129.391,396.021,164.523,60.727,160.585
C07027=1013.123,-129.141,396.013,164.526,60.725,160.585
C07028=1013.127,-128.892,396.004,164.528,60.722,160.585
C07029=1013.130,-128.642,395.996,164.531,60.718,160.585
C07030=1013.134,-128.393,395.989,164.533,60.714,160.585
C07031=1013.139,-128.143,395.982,164.535,60.710,160.585
C07032=1013.143,-127.893,395.976,164.538,60.706,160.585
C07033=1013.147,-127.644,395.969,164.539,60.701,160.585
C07034=1013.152,-127.394,395.963,164.542,60.697,160.585
C07035=1013.156,-127.144,395.956,164.545,60.692,160.585
C07036=1013.161,-126.894,395.950,164.547,60.688,160.585
C07037=1013.165,-126.645,395.942,164.549,60.683,160.585
C07038=1013.170,-126.395,395.936,164.551,60.679,160.585
C07039=1013.174,-126.144,395.930,164.554,60.675,160.585
C07040=1013.179,-125.894,395.923,164.556,60.670,160.584
C07041=1013.183,-125.645,395.916,164.559,60.666,160.584
C07042=1013.188,-125.395,395.910,164.560,60.661,160.584
C07043=1013.192,-125.145,395.903,164.564,60.656,160.584
C07044=1013.197,-124.895,395.896,164.566,60.652,160.584
C07045=1013.201,-124.645,395.890,164.568,60.647,160.584
C07046=1013.205,-124.395,395.882,164.570,60.643,160.584
C07047=1013.210,-124.145,395.876,164.574,60.638,160.584
C07048=1013.214,-123.895,395.870,164.575,60.633,160.584
C07049=1013.219,-123.646,395.862,164.577,60.629,160.584
C07050=1013.223,-123.396,395.856,164.580,60.624,160.583
C07051=1013.228,-123.146,395.849,164.583,60.620,160.583
C07052=1013.232,-122.896,395.842,164.584,60.615,160.583
C07053=1013.237,-122.646,395.835,164.588,60.610,160.583
C07054=1013.241,-122.396,395.829,164.590,60.606,160.583
C07055=1013.245,-122.146,395.822,164.592,60.601,160.583
C07056=1013.250,-121.897,395.815,164.595,60.597,160.583
C07057=1013.254,-121.646,395.808,164.597,60.592,160.583
C07058=1013.259,-121.397,395.801,164.599,60.586,160.582
C07059=1013.263,-121.147,395.795,164.602,60.582,160.582
C07060=1013.268,-120.897,395.787,164.603,60.577,160.582
C07061=1013.272,-120.647,395.780,164.607,60.573,160.582
C07062=1013.277,-120.398,395.774,164.608,60.568,160.582
C07063=1013.281,-120.148,395.767,164.612,60.563,160.582
C07064=1013.285,-119.898,395.760,164.613,60.558,160.582
C07065=1013.290,-119.648,395.752,164.616,60.553,160.581
C07066=1013.294,-119.398,395.746,164.619,60.549,160.581
C07067=1013.299,-119.148,395.739,164.621,60.543,160.581
C07068=1013.303,-118.898,395.732,164.624,60.539,160.581
C07069=1013.308,-118.617,395.725,164.626,60.533,160.581
C07070=1013.313,-118.336,395.716,164.628,60.528,160.581
C07071=1013.318,-118.056,395.709,164.631,60.522,160.580
C07072=1013.323,-117.775,395.701,164.634,60.517,160.580
C07073=1013.328,-117.526,395.694,164.637,60.512,160.580
C07074=1013.332,-117.276,395.686,164.639,60.508,160.580
C07075=1013.337,-117.025,395.680,164.642,60.502,160.580
C07076=1013.342,-116.776,395.672,164.643,60.497,160.580
C07077=1013.346,-116.526,395.665,164.646,60.492,160.579
C07078=1013.350,-116.276,395.658,164.649,60.487,160.580
C07079=1013.355,-116.026,395.651,164.651,60.483,160.579
C07080=1013.360,-115.777,395.644,164.654,60.477,160.579
C07081=1013.364,-115.527,395.637,164.656,60.472,160.579
C07082=1013.369,-115.276,395.630,164.658,60.467,160.579
C07083=1013.374,-115.027,395.623,164.662,60.462,160.579
C07084=1013.378,-114.777,395.615,164.663,60.457,160.578
C07085=1013.382,-114.527,395.609,164.666,60.452,160.578
C07086=1013.386,-114.277,395.601,164.668,60.447,160.578
C07087=1013.391,-114.028,395.594,164.670,60.442,160.578
C07088=1013.396,-113.777,395.586,164.673,60.437,160.578
C07089=1013.400,-113.528,395.579,164.676,60.432,160.578
C07090=1013.404,-113.278,395.572,164.678,60.427,160.577
C07091=1013.409,-113.028,395.565,164.681,60.422,160.577
C07092=1013.414,-112.779,395.558,164.683,60.417,160.577
C07093=1013.419,-112.528,395.550,164.685,60.411,160.577
C07094=1013.423,-112.279,395.543,164.688,60.406,160.577
C07095=1013.427,-112.029,395.535,164.690,60.401,160.576
C07096=1013.431,-111.779,395.529,164.693,60.396,160.576
C07097=1013.436,-111.528,395.521,164.695,60.391,160.576
C07098=1013.441,-111.279,395.513,164.697,60.386,160.575
C07099=1013.446,-111.029,395.507,164.700,60.380,160.575
C07100=1013.450,-110.780,395.499,164.702,60.375,160.575
C07101=1013.455,-110.529,395.491,164.705,60.370,160.575
C07102=1013.459,-110.280,395.484,164.707,60.365,160.575
C07103=1013.464,-110.030,395.477,164.710,60.359,160.574
C07104=1013.468,-109.780,395.470,164.712,60.354,160.574
C07105=1013.473,-109.530,395.462,164.715,60.349,160.574
C07106=1013.477,-109.280,395.455,164.718,60.343,160.574
C07107=1013.482,-109.030,395.447,164.720,60.339,160.574
C07108=1013.487,-108.781,395.441,164.722,60.333,160.573
C07109=1013.492,-108.531,395.433,164.725,60.328,160.573
C07110=1013.496,-108.281,395.425,164.727,60.322,160.573
C07111=1013.500,-108.031,395.418,164.730,60.316,160.573
C07112=1013.505,-107.781,395.410,164.733,60.311,160.573
C07113=1013.510,-107.531,395.403,164.734,60.306,160.572
C07114=1013.514,-107.282,395.395,164.737,60.301,160.572
C07115=1013.519,-107.032,395.388,164.740,60.296,160.572
C07116=1013.523,-106.782,395.380,164.743,60.290,160.572
C07117=1013.528,-106.532,395.373,164.745,60.284,160.571
C07118=1013.533,-106.282,395.365,164.747,60.279,160.571
C07119=1013.537,-106.032,395.358,164.749,60.274,160.571
C07120=1013.542,-105.783,395.350,164.752,60.269,160.570
C07121=1013.546,-105.533,395.341,164.755,60.263,160.570
C07122=1013.550,-105.283,395.334,164.757,60.258,160.570
C07123=1013.555,-105.033,395.326,164.759,60.252,160.570
C07124=1013.560,-104.783,395.319,164.762,60.246,160.570
C07125=1013.564,-104.533,395.311,164.765,60.241,160.569
C07126=1013.569,-104.283,395.303,164.768,60.236,160.569
C07127=1013.573,-104.034,395.295,164.770,60.230,160.569
C07128=1013.578,-103.784,395.288,164.771,60.225,160.568
C07129=1013.583,-103.534,395.280,164.774,60.220,160.568
C07130=1013.587,-103.284,395.273,164.777,60.214,160.568
C07131=1013.592,-103.034,395.265,164.779,60.208,160.568
C07132=1013.597,-102.785,395.257,164.782,60.203,160.567
C07133=1013.602,-102.504,395.249,164.785,60.196,160.567
C07134=1013.607,-102.224,395.240,164.787,60.190,160.567
C07135=1013.612,-101.943,395.231,164.790,60.184,160.566
C07136=1013.617,-101.663,395.222,164.793,60.177,160.566
C07137=1013.622,-101.413,395.215,164.796,60.172,160.566
C07138=1013.627,-101.163,395.207,164.798,60.166,160.565
C07139=1013.631,-100.914,395.199,164.801,60.160,160.565
C07140=1013.636,-100.663,395.190,164.804,60.155,160.565
C07141=1013.640,-100.413,395.183,164.806,60.149,160.565
C07142=1013.645,-100.163,395.175,164.809,60.144,160.564
C07143=1013.649,-99.914,395.167,164.811,60.138,160.564
C07144=1013.654,-99.664,395.159,164.813,60.132,160.564
C07145=1013.659,-99.414,395.152,164.816,60.126,160.563
C07146=1013.663,-99.165,395.144,164.818,60.121,160.563
C07147=1013.668,-98.915,395.136,164.820,60.115,160.563
C07148=1013.673,-98.665,395.128,164.823,60.109,160.563
C07149=1013.677,-98.415,395.119,164.825,60.103,160.562
C07150=1013.682,-98.165,395.112,164.828,60.097,160.562
C07151=1013.687,-97.915,395.104,164.831,60.091,160.562
C07152=1013.692,-97.665,395.096,164.834,60.086,160.561
C07153=1013.696,-97.415,395.088,164.836,60.080,160.561
C07154=1013.701,-97.166,395.079,164.839,60.075,160.561
C07155=1013.704,-96.916,395.071,164.841,60.069,160.560
C07156=1013.710,-96.666,395.063,164.844,60.063,160.560
C07157=1013.714,-96.416,395.055,164.846,60.057,160.560
C07158=1013.719,-96.166,395.046,164.849,60.052,160.559
C07159=1013.723,-95.916,395.039,164.851,60.046,160.559
C07160=1013.728,-95.667,395.030,164.853,60.041,160.559
C07161=1013.732,-95.416,395.022,164.856,60.035,160.558
C07162=1013.737,-95.167,395.014,164.858,60.029,160.558
C07163=1013.742,-94.917,395.005,164.860,60.023,160.558
C07164=1013.746,-94.668,394.997,164.863,60.018,160.557
C07165=1013.751,-94.418,394.989,164.866,60.011,160.557
C07166=1013.755,-94.167,394.981,164.868,60.005,160.557
C07167=1013.760,-93.918,394.972,164.871,60.000,160.557
C07168=1013.764,-93.668,394.964,164.873,59.994,160.556
C07169=1013.769,-93.419,394.956,164.876,59.989,160.556
C07170=1013.774,-93.169,394.948,164.878,59.983,160.555
C07171=1013.778,-92.918,394.939,164.881,59.976,160.555
C07172=1013.783,-92.669,394.931,164.884,59.971,160.555
C07173=1013.788,-92.419,394.922,164.886,59.965,160.554
C07174=1013.793,-92.169,394.914,164.888,59.959,160.554
C07175=1013.797,-91.920,394.906,164.891,59.953,160.554
C07176=1013.802,-91.670,394.897,164.894,59.947,160.554
C07177=1013.807,-91.420,394.889,164.897,59.941,160.553
C07178=1013.811,-91.170,394.881,164.899,59.935,160.553
C07179=1013.816,-90.921,394.872,164.901,59.929,160.552
C07180=1013.821,-90.670,394.864,164.905,59.923,160.552
C07181=1013.825,-90.421,394.856,164.907,59.917,160.552
C07182=1013.830,-90.171,394.847,164.909,59.911,160.551
C07183=1013.834,-89.921,394.839,164.911,59.905,160.551
C07184=1013.839,-89.672,394.831,164.914,59.898,160.550
C07185=1013.844,-89.422,394.822,164.917,59.893,160.550
C07186=1013.848,-89.171,394.814,164.919,59.887,160.550
C07187=1013.853,-88.922,394.806,164.922,59.880,160.549
C07188=1013.858,-88.672,394.797,164.924,59.874,160.549
C07189=1013.863,-88.422,394.788,164.926,59.868,160.548
C07190=1013.868,-88.172,394.780,164.930,59.862,160.548
C07191=1013.872,-87.923,394.772,164.932,59.856,160.548
C07192=1013.877,-87.673,394.763,164.934,59.850,160.547
C07193=1013.882,-87.423,394.754,164.937,59.843,160.547
C07194=1013.887,-87.173,394.746,164.939,59.837,160.546
C07195=1013.891,-86.924,394.738,164.941,59.831,160.546
C07196=1013.896,-86.674,394.729,164.945,59.824,160.546
C07197=1013.902,-86.395,394.720,164.948,59.818,160.545
C07198=1013.907,-86.116,394.710,164.950,59.811,160.545
C07199=1013.912,-85.838,394.700,164.954,59.804,160.544
C07200=1013.918,-85.560,394.691,164.956,59.797,160.544
C07201=1013.921,-85.310,394.683,164.958,59.791,160.543
C07202=1013.927,-85.060,394.675,164.961,59.784,160.543
C07203=1013.931,-84.810,394.665,164.964,59.778,160.543
C07204=1013.936,-84.560,394.657,164.967,59.772,160.542
C07205=1013.942,-84.311,394.648,164.968,59.765,160.541
C07206=1013.946,-84.061,394.640,164.971,59.759,160.541
C07207=1013.951,-83.811,394.632,164.974,59.753,160.541
C07208=1013.955,-83.561,394.623,164.977,59.746,160.540
C07209=1013.960,-83.311,394.614,164.979,59.740,160.540
C07210=1013.965,-83.061,394.605,164.982,59.733,160.540
C07211=1013.970,-82.812,394.597,164.984,59.727,160.539
C07212=1013.975,-82.562,394.589,164.987,59.720,160.539
C07213=1013.979,-82.312,394.580,164.989,59.714,160.538
C07214=1013.985,-82.063,394.571,164.992,59.708,160.538
C07215=1013.989,-81.813,394.562,164.994,59.701,160.537
C07216=1013.994,-81.563,394.554,164.997,59.694,160.537
C07217=1013.999,-81.313,394.546,164.999,59.688,160.536
C07218=1014.003,-81.063,394.537,165.002,59.682,160.536
C07219=1014.009,-80.814,394.529,165.005,59.675,160.535
C07220=1014.013,-80.564,394.520,165.007,59.669,160.535
C07221=1014.018,-80.314,394.511,165.010,59.662,160.535
C07222=1014.023,-80.064,394.502,165.012,59.656,160.534
C07223=1014.027,-79.814,394.493,165.016,59.650,160.534
C07224=1014.033,-79.565,394.484,165.017,59.643,160.533
C07225=1014.038,-79.315,394.475,165.020,59.636,160.533
C07226=1014.042,-79.065,394.466,165.022,59.630,160.532
C07227=1014.047,-78.815,394.456,165.026,59.624,160.532
C07228=1014.052,-78.565,394.448,165.028,59.618,160.531
C07229=1014.056,-78.315,394.439,165.030,59.611,160.531
C07230=1014.061,-78.065,394.430,165.032,59.605,160.530
C07231=1014.066,-77.816,394.421,165.036,59.598,160.530
C07232=1014.071,-77.566,394.412,165.038,59.592,160.530
C07233=1014.075,-77.316,394.403,165.040,59.585,160.529
C07234=1014.080,-77.067,394.394,165.044,59.578,160.529
C07235=1014.085,-76.817,394.385,165.046,59.572,160.528
C07236=1014.090,-76.567,394.375,165.048,59.565,160.528
C07237=1014.094,-76.317,394.366,165.051,59.559,160.527
C07238=1014.099,-76.067,394.358,165.054,59.553,160.527
C07239=1014.104,-75.817,394.349,165.055,59.546,160.526
C07240=1014.108,-75.567,394.340,165.059,59.539,160.526
C07241=1014.114,-75.318,394.331,165.061,59.532,160.525
C07242=1014.118,-75.068,394.321,165.063,59.526,160.525
C07243=1014.123,-74.818,394.312,165.066,59.520,160.524
C07244=1014.128,-74.568,394.303,165.069,59.512,160.524
C07245=1014.132,-74.319,394.294,165.071,59.506,160.523
C07246=1014.137,-74.069,394.284,165.074,59.500,160.523
C07247=1014.142,-73.819,394.275,165.077,59.494,160.522
C07248=1014.146,-73.569,394.266,165.079,59.487,160.522
C07249=1014.151,-73.320,394.256,165.081,59.481,160.521
C07250=1014.156,-73.069,394.246,165.085,59.474,160.521
C07251=1014.161,-72.820,394.237,165.087,59.468,160.521
C07252=1014.166,-72.570,394.227,165.089,59.461,160.520
C07253=1014.170,-72.320,394.218,165.092,59.455,160.519
///RCONF 1,0,0,0,0,0,0,0,0,0,0,0,0,0,0,0,0,0,0,0,0,0,0,0
C07254=1014.175,-72.070,394.209,165.095,59.448,160.519
C07255=1014.180,-71.821,394.199,165.096,59.442,160.518
C07256=1014.184,-71.571,394.190,165.100,59.435,160.518
C07257=1014.189,-71.322,394.180,165.103,59.429,160.518
C07258=1014.194,-71.071,394.171,165.104,59.422,160.517
C07259=1014.198,-70.822,394.161,165.108,59.416,160.517
C07260=1014.203,-70.572,394.152,165.109,59.409,160.516
C07261=1014.209,-70.296,394.142,165.113,59.401,160.515
C07262=1014.214,-70.019,394.131,165.115,59.394,160.515
C07263=1014.219,-69.742,394.120,165.118,59.387,160.514
C07264=1014.224,-69.466,394.109,165.121,59.380,160.514
C07265=1014.229,-69.216,394.100,165.124,59.373,160.513
C07266=1014.234,-68.966,394.090,165.126,59.366,160.513
C07267=1014.238,-68.716,394.081,165.129,59.360,160.512
C07268=1014.243,-68.467,394.071,165.131,59.353,160.512
C07269=1014.248,-68.217,394.062,165.134,59.346,160.511
C07270=1014.253,-67.967,394.052,165.136,59.339,160.511
C07271=1014.258,-67.717,394.042,165.139,59.333,160.510
C07272=1014.262,-67.467,394.033,165.142,59.326,160.510
C07273=1014.267,-67.218,394.023,165.144,59.320,160.509
C07274=1014.272,-66.968,394.014,165.147,59.313,160.509
